(* CODESYS project Plc_CHALET_Nc.library
   Placeholder: CHALET_Nc
   Title: CHALET_Nc
   Version: 3.4.2
   Company: Beckhoff CH

Project tree, tasks and I/O mapping:
  libraries: CHALET_BaseComponents, * (Beckhoff CH); Tc2_MC2, * (Beckhoff Automation GmbH); Tc2_MC2_Drive, * (Beckhoff Automation GmbH); Tc2_Standard, * (Beckhoff Automation GmbH); Tc2_System, * (Beckhoff Automation GmbH); Tc3_EventLogger, * (Beckhoff Automation GmbH); Tc3_Module, * (Beckhoff Automation GmbH)
  COMPONENTs/
    Main FB/
      function block FB_NcAxis [ST]: Mapped, NcAxisName, NcAxisType, NcDriveType, NetId, OID, Port, GearIn, GearOut, Homing, HomingSensor, LockNegativeDirection, LockPositiveDirection, MoveAbsolute, MoveRelative, MoveVelocity, MultiGearIn, PowerOff, PowerOn, Reset, SetActPosition, Stop, ActAcceleration, ActPosition, ActPosModulo, ActVelocity, DefaultAcceleration, DefaultDeceleration, DefaultJerk, DefaultVelocity, Override, SetAcceleration, SetPosition, SetPosModulo, SetVelocity, BufferEmpty, Coupled, Enabled, Feedback, LagDistance, MotionState, Moving, FB_init, Initialize, Initialized, Prepare, Update
      interface I_AxisStatus: Override, SetAcceleration, SetPosition, SetPosModulo, SetVelocity, Enabled, LagDistance, LockNegativeDirection, LockPositiveDirection, Mapped, MotionState, Feedback, Initialized
      interface I_NcAxis_HMI: Coupled, LUID, Moving, NcAxisName
      interface I_NcAxis_PLC: GearIn, GearOut, Homing, LockNegativeDirection, LockPositiveDirection, MoveAbsolute, MoveRelative, MoveVelocity, MultiGearIn, PowerOff, PowerOn, Reset, SetActPosition, Stop, ActAcceleration, ActPosition, ActPosModulo, ActVelocity, DefaultAcceleration, DefaultDeceleration, DefaultJerk, DefaultVelocity, Override, BufferEmpty, NcAxisType, NcDriveType, Initialize, Update
    Optional/
      Adapter AXIS_REF/
        function block FB_Adapter_AXIS_REF [ST]: getAxisRef
        interface I_Adapter_AXIS_REF: getAxisRef
      Adapter HMI/
        function block FB_NcAxis_Hmi [ST]: FB_init, Update
      Casting/
        function ToNcAxisHMI [ST]
        function ToNcAxisPLC [ST]
      Feedback/
        function block FB_NcFeedback [ST]: UpdateEventlogger
      Reset/
        function block FB_Reset_NC_Sercos_CANopen [ST]
      SetActPosition/
        old/
          function block FB_SetPosition_NC_Sercos_CANopen [ST]: SetPosCoE, SetPosNC, SetPosSoE
        function block FB_SetPosition_Beckhoff [ST]
    data type E_NcAxisCommands
    NcAxisFB
  00000000-0000-0000-0000-000000000000|LICENSE.md
  LICENSE.md
  global variables NcParameterlist
*)

// COMPONENTs/E_NcAxisCommands
{attribute 'strict'}
{attribute 'to_string'}
TYPE E_NcAxisCommands :
(
	None:=0,
	Initialize,
	Reset,
	PowerOn,
	PowerOff,
	SetPosition,
	Stop,
	MoveVelocity,
	MoveRelative,
	MoveAbsolute,
	GearIn,
	GearOut,
	MultiGearIn,
	Homing,
	
	//Commands that are not handled within the basic module and must be implemented externally
	TorqueControl:=100,
	Halt,
	Jog,
	GearInDyn,
	MoveModulo,
	HaltPhasing,
	PhasingAbsolute,
	PhasingRelative,
	MoveContinuousAbsolute,
	MoveContinuousRelative,
	MoveSuperImposed,
	AbortSuperposition,
	MoveAbsoluteCA,
	MoveRelativeCA,
	HaltCA,
	GearInPosCA,
	StartExternalSetpoint,
	StopExternalSetpoint,
	
	//xPlanar
	Enable,
	Disable,
	AddToGroupe,
	RemoveFromGroupe,
	Configure,
	MoveA,
	MoveB,
	MoveC,
	MoveXY,
	MoveZ,
	JoinTrack,
	MoveOnTrack,
	Clear,
	LowerToUnknownLevel,
	LiftFromUnknownLevel,
	
	
	//Reserve
	ExternalCommand00:=200,	
	ExternalCommand01,
	ExternalCommand02,
	ExternalCommand03,
	ExternalCommand04,
	ExternalCommand05,
	ExternalCommand06,
	ExternalCommand07,
	ExternalCommand08,
	ExternalCommand09,
	ExternalCommand10,	
	ExternalCommand11,
	ExternalCommand12,
	ExternalCommand13,
	ExternalCommand14,
	ExternalCommand15,
	ExternalCommand16,
	ExternalCommand17,
	ExternalCommand18,
	ExternalCommand19

//default is none	
) := None;
END_TYPE

// NcParameterlist
{attribute 'qualified_only'}
VAR_GLOBAL CONSTANT
	ERROR_IF_NC_AXIS_IS_NOT_MAPPED : BOOL := TRUE;
END_VAR

// COMPONENTs/Main FB/FB_NcAxis
// The warning " Interface of overridden methode xxx of base I_xxx doesn't match declaration" can be disabled here. 
{warning disable C0094 }
{attribute 'no_explicit_call' := '[FB_NcAxis] Do not call the body - Stick to OOP'}
FUNCTION_BLOCK FB_NcAxis EXTENDS FB_Adapter_AXIS_REF IMPLEMENTS I_NcAxis_PLC, I_NcAxis_HMI, I_AdsAddr
VAR
	{attribute 'hide'}
	bInitDone : BOOL;
	
	//Default Values is used if commandet jerk, acc, dec or velo is 0.
	{attribute 'hide'}
	fDefaultVelocity 		: LREAL; // Read during init from NC-Axis-Parameter(init)
	{attribute 'hide'}
	fDefaultAcceleration 	: LREAL; // Read during init from NC-Axis-Parameter(init)
	{attribute 'hide'}
	fDefaultDeceleration	: LREAL; // Read during init from NC-Axis-Parameter(init)
	{attribute 'hide'}
	fDefaultJerk 			: LREAL; // Read during init from NC-Axis-Parameter(init)	
	
	//Full axis parameter set
	{attribute 'hide'}
	stAxisParameterSet 		: TC2_MC2.ST_AxisParameterSet;
	
	//Velocity override in % for all movement commands. (0 ≤ Override ≤ 100.0)
	{attribute 'hide'}
	fOverride : LREAL := 100.0;
	//Feed enable in x direction. Only takes effect if Enable = TRUE.
	{attribute 'hide'}
	bLockNegativeDirection : BOOL := FALSE;
	{attribute 'hide'}
	bLockPositiveDirection : BOOL := FALSE;
	
	//GearIn
	{attribute 'hide'}
	ipGearMasterAxis 		: I_Adapter_AXIS_REF;

	//Multigear
	{attribute 'hide'}
	ipMultiGearMasterAxis1		: I_Adapter_AXIS_REF;
	{attribute 'hide'}
	ipMultiGearMasterAxis2		: I_Adapter_AXIS_REF;
	{attribute 'hide'}
	ipMultiGearMasterAxis3		: I_Adapter_AXIS_REF;
	{attribute 'hide'}
	ipMultiGearMasterAxis4		: I_Adapter_AXIS_REF;

	{attribute 'hide'}
	fbDummyAxisRef		: TC2_MC2.AXIS_REF; // AxisRef whitout linked Nc
	
	{attribute 'hide'}               	
	fbFeedback 			: FB_NcFeedback(ipSourceInfo := fbSourceInfo);	
	
 	{attribute 'hide'}                   	
	eActiveCommand 		: E_NcAxisCommands := E_NcAxisCommands.None;
	
	{attribute 'hide'}           	
	fbPower 			: MC_Power;
	{attribute 'hide'}
	fbStop 				: MC_Stop;
	{attribute 'hide'}
	fbHoming 			: MC_Home;
	{attribute 'hide'}
	fbReset 			: FB_Reset_NC_Sercos_CANopen; 		//MC_Reset extension. can detect sercos and can and reset all faults.
	{attribute 'hide'}
	fbSetPosition 		: FB_SetPosition_Beckhoff;	//MC_SetPosition extension. Detect sercos and can and read and use the configured store position of the position feedback.(encoder/drive/NC). Set store position in DM2.
	{attribute 'hide'}
	fbMoveRelative 		: ARRAY [0..1] OF MC_MoveRelative;//A second function block is always required to use the BufferMode. It is not possible to trigger a move function block with new parameters while it is active.
	{attribute 'hide'}
	nActiveMoveRel		: UINT; 
	{attribute 'hide'}
	fbMoveAbsolute		: ARRAY [0..1] OF MC_MoveAbsolute;//A second function block is always required to use the BufferMode. It is not possible to trigger a move function block with new parameters while it is active.
	{attribute 'hide'}
	nActiveMoveAbs		: UINT; 
	{attribute 'hide'}
	fbMoveVelocity		: ARRAY [0..1] OF MC_MoveVelocity;//A second function block is always required to use the BufferMode. It is not possible to trigger a move function block with new parameters while it is active.
	{attribute 'hide'}
	nActiveMoveVel		: UINT; 
	{attribute 'hide'}
	fbGearInMultiMaster	: MC_GearInMultiMaster;
	{attribute 'hide'}
	fbGearIn 			: MC_GearIn;
	{attribute 'hide'}
	fbGearOut 			: MC_GearOut;

	{attribute 'hide'}
	bNewBufferCommadThisCycle : BOOL; //This flag is processed in the PLC cycle when a buffered motion command is requested via method


END_VAR
{warning restore C0094}

{attribute 'monitoring':='call'}
PROPERTY Mapped : BOOL //Project is mapped to NC (NcToPlc and PlcToNc)
GET
VAR
	bNcToPlcNotMapped 	: BOOL;
	bPlcToNcNotMapped 	: BOOL;
END_VAR
bPlcToNcNotMapped := F_GetMappingStatus(ADR(THIS^.Axis.PlcToNc), SIZEOF(THIS^.Axis.PlcToNc)) <> EPlcMappingStatus.MS_Mapped;
bNcToPlcNotMapped := F_GetMappingStatus(ADR(THIS^.Axis.NcToPlc), SIZEOF(THIS^.Axis.NcToPlc)) <> EPlcMappingStatus.MS_Mapped;

Mapped := NOT bNcToPlcNotMapped AND NOT bPlcToNcNotMapped;
END_GET
END_PROPERTY

{attribute 'OPC.UA.DA.Property' := '1'}
{attribute 'monitoring':='call'}
PROPERTY NcAxisName : String(31)
GET
NcAxisName := THIS^.stAxisParameterSet.sAxisName;
END_GET
END_PROPERTY

{attribute 'OPC.UA.DA.Property' := '1'}
{attribute 'monitoring':='call'}
PROPERTY NcAxisType : Tc2_MC2.E_NcAxisType
GET
NcAxisType := THIS^.stAxisParameterSet.nAxisType;
END_GET
END_PROPERTY

{attribute 'OPC.UA.DA.Property' := '1'}
{attribute 'monitoring':='call'}
PROPERTY NcDriveType : Tc2_MC2.E_NcDriveType
GET
NcDriveType:= THIS^.Axis.DriveAddress.NcDriveType;
END_GET
END_PROPERTY

{attribute 'monitoring':='call'}
PROPERTY NetId : T_AmsNetID
GET
NetId := THIS^.Axis.DriveAddress.NetID;
END_GET
END_PROPERTY

{attribute 'monitoring':='call'}
PROPERTY OID : OTCID
GET
OID := THIS^.Axis.DriveAddress.TcAxisObjectId;
END_GET
END_PROPERTY

{attribute 'monitoring':='call'}
PROPERTY Port : WORD
GET
Port := THIS^.Axis.DriveAddress.SlaveAddress;
END_GET
END_PROPERTY

{attribute 'TcRpcEnable':='1'}
(*! 
<summary>
	Establish an axis coupling to a single master axis.
	<preliminary>
		Both axis must be in standstill to apply the coupling.
		In-motion coupling of the FB is not supported by this method.
	</preliminary>
</summary>
<description>
	The coupling is performed based on a <b>velocity</b> ratio.
	As reference the master axis <b>command</b> value is used.
	There is <b>no automatic phase compensation</b> applied.
</description> 
*)

METHOD PUBLIC GearIn  : I_CH_Feedback (*! Interface to the execution feedback *)
VAR_INPUT
	(*! Interface to a master axis *)
	ipMasterAxisAdapter : I_Adapter_AXIS_REF;

	(*! Gear ratio Numerator*)
	fRatioNumerator: LREAL;
	
	(*! Gear ratio Denominator*)
	nRatioDenominator: UINT := 1;
	
	(*! Use the default dynamics if input=0.
	The default dynamics can be read and written via property and is initialized with the default values in the NC parameter list. *)
	fAcceleration	: LREAL := 0;
	
	(*! Use the default dynamics if input=0. 
	The default dynamics can be read and written via property and is initialized with the default values in the NC parameter list. *)
	fDeceleration	: LREAL := 0;
	
	(*! Use the default dynamics if input=0. 
	The default dynamics can be read and written via property and is initialized with the default values in the NC parameter list. *)
	fJerk			: LREAL := 0;
END_VAR
IF ipMasterAxisAdapter = 0 THEN
	THIS^.fbFeedback.LastCommandAccepted	:= FALSE;
	//Error not valid Input
	
ELSIF NOT __ISVALIDREF(ipMasterAxisAdapter.getAxisRef) THEN
	THIS^.fbFeedback.LastCommandAccepted	:= FALSE;
	//Invalide ref to axis
	
ELSIF fRatioNumerator = 0 OR nRatioDenominator = 0 THEN
	THIS^.fbFeedback.LastCommandAccepted	:= FALSE;
	//Error not valid Input		
	
ELSIF THIS^.fbFeedback.Error THEN
	THIS^.fbFeedback.LastCommandAccepted	:= FALSE;
	//Error active/not ready

ELSIF ipMasterAxisAdapter.getAxisRef.Status.Moving THEN		
	THIS^.fbFeedback.LastCommandAccepted	:= FALSE;
	//Only support geraring in standstill

ELSIF THIS^.Axis.Status.Moving THEN		
	THIS^.fbFeedback.LastCommandAccepted	:= FALSE;	
	//Only support geraring in standstill

ELSE
	THIS^.eActiveCommand 				:= E_NcAxisCommands.GearIn;
	THIS^.fbFeedback.ActiveCommand 		:= TO_STRING(THIS^.eActiveCommand);
	THIS^.fbFeedback.LastCommandAccepted:= TRUE;
	THIS^.fbFeedback.Busy 				:= TRUE;
	
	THIS^.ipGearMasterAxis 				:= ipMasterAxisAdapter;
	
	THIS^.fbGearIn.Execute				:= TRUE;
	THIS^.fbGearIn.RatioNumerator 		:= fRatioNumerator;	
	THIS^.fbGearIn.RatioDenominator     := nRatioDenominator;		
	
	//Acceleration
	//If input = 0  then use default dynamics
	IF fAcceleration = 0.0 THEN
		THIS^.fbGearIn.Acceleration := THIS^.fDefaultAcceleration;
	ELSE
		THIS^.fbGearIn.Acceleration := fAcceleration;
	END_IF
	
	//Deceleration
	//If input = 0  then use default dynamics
	IF fDeceleration = 0.0 THEN
		THIS^.fbGearIn.Deceleration := THIS^.fDefaultDeceleration;
	ELSE
		THIS^.fbGearIn.Deceleration := fDeceleration;
	END_IF
	
	//Jerk
	//If input = 0  then use default dynamics
	IF fJerk = 0.0 THEN
		THIS^.fbGearIn.Jerk := THIS^.fDefaultJerk;
	ELSE
		THIS^.fbGearIn.Jerk := fJerk;
	END_IF
END_IF


GearIn := THIS^.fbFeedback;
END_METHOD

{attribute 'TcRpcEnable':='1'} 
(*WARNING
No standstill of the axis due to decoupling
When a slave axis is uncoupled during the movement, it is not stopped automatically but reaches a constant velocity at which it continues to travel infinitely.
You can stop the axis with the function blocks MC_Halt or MC_Stop.*)
METHOD GearOut  : I_CH_Feedback


THIS^.eActiveCommand 				:= E_NcAxisCommands.GearOut;
THIS^.fbFeedback.ActiveCommand 		:= TO_STRING(THIS^.eActiveCommand);
THIS^.fbFeedback.LastCommandAccepted:= TRUE;
THIS^.fbFeedback.Busy 				:= TRUE;

THIS^.fbGearOut.Execute				:= TRUE;

THIS^.ipGearMasterAxis 				:= 0;
THIS^.ipMultiGearMasterAxis1 		:= 0;
THIS^.ipMultiGearMasterAxis2 		:= 0;
THIS^.ipMultiGearMasterAxis3 		:= 0;
THIS^.ipMultiGearMasterAxis4 		:= 0;



GearOut := THIS^.fbFeedback;
END_METHOD

{attribute 'TcRpcEnable':='1'} 
(*The parameterization of the home command takes place in the NC! To do this, set the parameters in:
- NC-Axis(Parameters) Homing speed
- NC-Axis>Encoder(Parameters) Homing mode
	Reference Mode: "Homing Sensor Only"
	Homing Sensor Source "Digital Input x" 
		Link Input to NC-Axis>Drive>Inputs>nState8.x
		
The "HomeingSensor" property can also be used to control a home sensor via PLC.		
*)
(*Homing refers to an axis initialization run during which the correct actual position is determined by means of a reference signal. This can be NC-guided, as default described here:
  - The axis is at a random position.
  - The axis moves in the parameterized direction and searches for the reference switch (referencing cam/calibration cam).
  - The axis reverses as soon as the referencing cam is detected.
  - The axis moves away from the referencing cam and detects the falling edge of the cam signal.
  - The reference position is set and the axis stops. The standstill position of the axis deviates slightly from the reference position.*)
METHOD Homing  : I_CH_Feedback
VAR_INPUT
	(*Absolute reference position to which the axis is set after homing*)
	fPosition		: LREAL;
END_VAR
IF THIS^.fbFeedback.Error THEN
	THIS^.fbFeedback.LastCommandAccepted	:= FALSE;
	//Error active/not ready

ELSIF NOT THIS^.BufferEmpty THEN		
	THIS^.fbFeedback.LastCommandAccepted	:= FALSE;
	//Buffer not ready to store next motion command	
	
ELSIF NOT(THIS^.Axis.Status.StandStill OR THIS^.Axis.Status.DiscreteMotion OR THIS^.Axis.Status.ContinuousMotion OR THIS^.Axis.Status.SynchronizedMotion) THEN		
	THIS^.fbFeedback.LastCommandAccepted	:= FALSE;
	//Axis in wrong State

	
ELSE
	THIS^.eActiveCommand 				:= E_NcAxisCommands.Homing;
	THIS^.fbFeedback.ActiveCommand 		:= TO_STRING(THIS^.eActiveCommand);
	THIS^.fbFeedback.LastCommandAccepted:= TRUE;                                  
	THIS^.fbFeedback.Busy 				:= TRUE;
	                                    
	THIS^.fbHoming.Execute				:= TRUE;
	 (* default homing as defined in the SystemManager encoder parameters *)
	THIS^.fbHoming.HomingMode			:= MC_HomingMode.MC_DefaultHoming;
	
	THIS^.fbHoming.Position				:= fPosition;
	
END_IF


Homing := THIS^.fbFeedback;
END_METHOD

//A home input switch can be linked here. Whether this works depends heavily on how the settings in the NC2-axis and NC2-axis-encoder are configured.
PROPERTY HomingSensor : BOOL
SET
THIS^.fbHoming.bCalibrationCam := HomingSensor;
END_SET
END_PROPERTY

{attribute 'monitoring':='call'}
//Disable the feed in one direction.
PROPERTY LockNegativeDirection : BOOL
GET
LockNegativeDirection := bLockNegativeDirection;
END_GET
SET
VAR_INST
	{attribute 'hide'}
	fbInfoFeedDisabled : FB_TcAlarm;
END_VAR
THIS^.bLockNegativeDirection := LockNegativeDirection;


//Creat an info in TC3_Eventlogger
IF NOT fbInfoFeedDisabled.bRaised AND THIS^.bLockNegativeDirection THEN
	fbInfoFeedDisabled.CreateEx(stEventEntry := TC_EVENTS.CHALET_NC_Events.FeedNegativeDisabled, bWithConfirmation := FALSE, ipSourceInfo := THIS^.fbSourceInfo);
	fbInfoFeedDisabled.Raise(0);
	
ELSIF NOT THIS^.bLockNegativeDirection THEN
	fbInfoFeedDisabled.Clear(0, 0);
END_IF
END_SET
END_PROPERTY

{attribute 'monitoring':='call'}
//Disable the feed in one direction.
PROPERTY LockPositiveDirection : BOOL
GET
LockPositiveDirection := bLockPositiveDirection;
END_GET
SET
VAR_INST
	{attribute 'hide'}
	fbInfoFeedDisabled : FB_TcAlarm;
END_VAR
THIS^.bLockPositiveDirection := LockPositiveDirection;


//Creat an info in TC3_Eventlogger
IF NOT fbInfoFeedDisabled.bRaised AND THIS^.bLockPositiveDirection THEN
	fbInfoFeedDisabled.CreateEx(stEventEntry := TC_EVENTS.CHALET_NC_Events.FeedPositiveDisabled, bWithConfirmation := FALSE, ipSourceInfo := THIS^.fbSourceInfo);
	fbInfoFeedDisabled.Raise(0);
	
ELSIF NOT THIS^.bLockPositiveDirection THEN
	fbInfoFeedDisabled.Clear(0, 0);
END_IF
END_SET
END_PROPERTY

{attribute 'TcRpcEnable':='1'} 
METHOD MoveAbsolute  : I_CH_Feedback
VAR_INPUT
	fPosition		: LREAL;
	
	(* Use the default dynamics if input=0. 
	The default dynamics can be read and written via property and is initialized with the default values in the NC parameter list. *)
	fVelocity		: LREAL := 0;
	
	(* Use the default dynamics if input=0. 
	The default dynamics can be read and written via property and is initialized with the default values in the NC parameter list. *)
	fAcceleration	: LREAL := 0;
	
	(* Use the default dynamics if input=0. 
	The default dynamics can be read and written via property and is initialized with the default values in the NC parameter list. *)
	fDeceleration	: LREAL := 0;
	
	(* Use the default dynamics if input=0. 
	The default dynamics can be read and written via property and is initialized with the default values in the NC parameter list. *)
	fJerk			: LREAL := 0;
	
	(* Input=0 = MC_Aborting   
	BufferModes:
		-MC_Aborting: Default mode without buffering. The command is executed immediately and interrupts any other command that may be running.
		-MC_Buffered: The command is executed once no other command is running on the axis. The previous movement continues until it has stopped. The following command is started from standstill.
		-MC_BlendingLow: The command is executed once no other command is running on the axis. In contrast to Buffered the axis does not stop at the previous target, but passes through this position with the lower velocity of two commands.
		-MC_BlendingHigh The command is executed once no other command is running on the axis. In contrast to Buffered the axis does not stop at the previous target, but passes through this position with the higher velocity of two commands.
		-MC_BlendingNext: The command is executed once no other command is running on the axis. In contrast to Buffered the axis does not stop at the previous target, but passes through this position with the velocity of the last command.
		-MC_BlendingPrevious: The command is executed once no other command is running on the axis. In contrast to Buffered the axis does not stop at the previous target, but passes through this position with the velocity of the first command. *)
	eBufferMode   : Tc2_MC2.MC_BufferMode := Tc2_MC2.MC_BufferMode.MC_Aborting;
END_VAR
VAR
	nInactiveInstance : UINT;
END_VAR
IF THIS^.fbFeedback.Error THEN
	THIS^.fbFeedback.LastCommandAccepted	:= FALSE;
	//Error active/not ready

ELSIF NOT THIS^.BufferEmpty THEN		
	THIS^.fbFeedback.LastCommandAccepted	:= FALSE;
	//Buffer not ready to store next motion command	
	
ELSIF NOT(THIS^.Axis.Status.StandStill OR THIS^.Axis.Status.DiscreteMotion OR THIS^.Axis.Status.ContinuousMotion OR THIS^.Axis.Status.SynchronizedMotion) THEN		
	THIS^.fbFeedback.LastCommandAccepted	:= FALSE;
	//Axis in wrong State
	
ELSIF (eBufferMode <> MC_BufferMode.MC_Aborting) AND bNewBufferCommadThisCycle THEN		
	THIS^.fbFeedback.LastCommandAccepted	:= FALSE;
	//Buffer not ready to store next motion command		
	//Max send one buffered motion command each cycle	
	
ELSE
	//A second function block is always required to use the BufferMode. It is not possible to trigger a move function block with new parameters while it is active.
	IF THIS^.fbMoveAbsolute[nActiveMoveAbs].Busy THEN
		nInactiveInstance := (THIS^.nActiveMoveAbs + 1)MOD 2;
	ELSE
		nInactiveInstance := THIS^.nActiveMoveAbs;
	END_IF
	
	THIS^.eActiveCommand 				:= E_NcAxisCommands.MoveAbsolute;
	THIS^.fbFeedback.ActiveCommand 		:= TO_STRING(THIS^.eActiveCommand);
	THIS^.fbFeedback.LastCommandAccepted:= TRUE;		
	THIS^.fbFeedback.Busy 				:= TRUE;
	
	THIS^.fbMoveAbsolute[nInactiveInstance].Execute		:= TRUE;
	THIS^.fbMoveAbsolute[nInactiveInstance].Position	:= fPosition;
	THIS^.fbMoveAbsolute[nInactiveInstance].BufferMode 	:= eBufferMode;
	
	//If the currend command is a buffered movement, then set a flag.
	IF eBufferMode <> MC_BufferMode.MC_Aborting THEN
		THIS^.bNewBufferCommadThisCycle := TRUE;
	END_IF
	
	//Velocity
	//If input = 0  then use default dynamics
	IF fVelocity = 0.0 THEN
		THIS^.fbMoveAbsolute[nInactiveInstance].Velocity := THIS^.fDefaultVelocity;
	ELSE
		THIS^.fbMoveAbsolute[nInactiveInstance].Velocity := fVelocity;
	END_IF
	
	//Acceleration
	//If input = 0  then use default dynamics
	IF fAcceleration = 0.0 THEN
		THIS^.fbMoveAbsolute[nInactiveInstance].Acceleration := THIS^.fDefaultAcceleration;
	ELSE
		THIS^.fbMoveAbsolute[nInactiveInstance].Acceleration := fAcceleration;
	END_IF
	
	//Deceleration
	//If input = 0  then use default dynamics
	IF fDeceleration = 0.0 THEN
		THIS^.fbMoveAbsolute[nInactiveInstance].Deceleration := THIS^.fDefaultDeceleration;
	ELSE
		THIS^.fbMoveAbsolute[nInactiveInstance].Deceleration := fDeceleration;
	END_IF
	
	//Jerk
	//If input = 0  then use default dynamics
	IF fJerk = 0.0 THEN
		THIS^.fbMoveAbsolute[nInactiveInstance].Jerk := THIS^.fDefaultJerk;
	ELSE
		THIS^.fbMoveAbsolute[nInactiveInstance].Jerk := fJerk;
	END_IF

END_IF


MoveAbsolute := THIS^.fbFeedback;
END_METHOD

{attribute 'TcRpcEnable':='1'} 
METHOD MoveRelative  : I_CH_Feedback
VAR_INPUT
	fDistance		: LREAL;
	
	(* Use the default dynamics if input=0. 
	The default dynamics can be read and written via property and is initialized with the default values in the NC parameter list. *)
	fVelocity		: LREAL := 0;
	
	(* Use the default dynamics if input=0. 
	The default dynamics can be read and written via property and is initialized with the default values in the NC parameter list. *)
	fAcceleration	: LREAL := 0;
	
	(* Use the default dynamics if input=0. 
	The default dynamics can be read and written via property and is initialized with the default values in the NC parameter list. *)
	fDeceleration	: LREAL := 0;
	
	(* Use the default dynamics if input=0. 
	The default dynamics can be read and written via property and is initialized with the default values in the NC parameter list. *)
	fJerk			: LREAL := 0;
	
	(* Input=0 = MC_Aborting   
	BufferModes:
		-MC_Aborting: Default mode without buffering. The command is executed immediately and interrupts any other command that may be running.
		-MC_Buffered: The command is executed once no other command is running on the axis. The previous movement continues until it has stopped. The following command is started from standstill.
		-MC_BlendingLow: The command is executed once no other command is running on the axis. In contrast to Buffered the axis does not stop at the previous target, but passes through this position with the lower velocity of two commands.
		-MC_BlendingHigh The command is executed once no other command is running on the axis. In contrast to Buffered the axis does not stop at the previous target, but passes through this position with the higher velocity of two commands.
		-MC_BlendingNext: The command is executed once no other command is running on the axis. In contrast to Buffered the axis does not stop at the previous target, but passes through this position with the velocity of the last command.
		-MC_BlendingPrevious: The command is executed once no other command is running on the axis. In contrast to Buffered the axis does not stop at the previous target, but passes through this position with the velocity of the first command. *)
	eBufferMode   : Tc2_MC2.MC_BufferMode := Tc2_MC2.MC_BufferMode.MC_Aborting;
END_VAR
VAR
	nInactiveInstance : UINT;
END_VAR
IF THIS^.fbFeedback.Error THEN
	THIS^.fbFeedback.LastCommandAccepted	:= FALSE;
	//Error active/not ready

ELSIF NOT THIS^.BufferEmpty THEN		
	THIS^.fbFeedback.LastCommandAccepted	:= FALSE;
	//Buffer not ready to store next motion command	
	
ELSIF NOT(THIS^.Axis.Status.StandStill OR THIS^.Axis.Status.DiscreteMotion OR THIS^.Axis.Status.ContinuousMotion OR THIS^.Axis.Status.SynchronizedMotion) THEN		
	THIS^.fbFeedback.LastCommandAccepted	:= FALSE;
	//Axis in wrong State

ELSIF (eBufferMode <> MC_BufferMode.MC_Aborting) AND bNewBufferCommadThisCycle THEN		
	THIS^.fbFeedback.LastCommandAccepted	:= FALSE;
	//Buffer not ready to store next motion command		
	//Max send one buffered motion command each cycle	
		
	
//ZZZ Todo Bug in 4024, only allow buffered movement if an 'normal' movement is active.	
ELSIF (eBufferMode <> MC_BufferMode.MC_Aborting) AND NOT THIS^.Axis.Status.HasJob THEN		
	THIS^.fbFeedback.LastCommandAccepted	:= FALSE;
	//Buffered movement not possible if axis is not moving
	
ELSE
	//A second function block is always required to use the BufferMode. It is not possible to trigger a move function block with new parameters while it is active.
	IF THIS^.fbMoveRelative[nActiveMoveRel].Busy THEN
		nInactiveInstance := (THIS^.nActiveMoveRel + 1)MOD 2;
	ELSE
		nInactiveInstance := THIS^.nActiveMoveRel;
	END_IF

	THIS^.eActiveCommand 				:= E_NcAxisCommands.MoveRelative;
	THIS^.fbFeedback.ActiveCommand 		:= TO_STRING(THIS^.eActiveCommand);
	THIS^.fbFeedback.LastCommandAccepted:= TRUE;                                  
	THIS^.fbFeedback.Busy 				:= TRUE;
	                                    
	THIS^.fbMoveRelative[nInactiveInstance].Execute		:= TRUE;
	THIS^.fbMoveRelative[nInactiveInstance].Distance	:= fDistance;
	THIS^.fbMoveRelative[nInactiveInstance].BufferMode 	:= eBufferMode;
	
	//If the currend command is a buffered movement, then set a flag.
	IF eBufferMode <> MC_BufferMode.MC_Aborting THEN
		THIS^.bNewBufferCommadThisCycle := TRUE;
	END_IF
	
	//Velocity
	//If input = 0  then use default dynamics
	IF fVelocity = 0.0 THEN
		THIS^.fbMoveRelative[nInactiveInstance].Velocity := THIS^.fDefaultVelocity;
	ELSE
		THIS^.fbMoveRelative[nInactiveInstance].Velocity := fVelocity;
	END_IF
	
	//Acceleration
	//If input = 0  then use default dynamics
	IF fAcceleration = 0.0 THEN
		THIS^.fbMoveRelative[nInactiveInstance].Acceleration := THIS^.fDefaultAcceleration;
	ELSE
		THIS^.fbMoveRelative[nInactiveInstance].Acceleration := fAcceleration;
	END_IF
	
	//Deceleration
	//If input = 0  then use default dynamics
	IF fDeceleration = 0.0 THEN
		THIS^.fbMoveRelative[nInactiveInstance].Deceleration := THIS^.fDefaultDeceleration;
	ELSE
		THIS^.fbMoveRelative[nInactiveInstance].Deceleration := fDeceleration;
	END_IF
	
	//Jerk
	//If input = 0  then use default dynamics
	IF fJerk = 0.0 THEN
		THIS^.fbMoveRelative[nInactiveInstance].Jerk := THIS^.fDefaultJerk;
	ELSE
		THIS^.fbMoveRelative[nInactiveInstance].Jerk := fJerk;
	END_IF
END_IF


MoveRelative := THIS^.fbFeedback;
END_METHOD

{attribute 'TcRpcEnable':='1'} 
METHOD MoveVelocity  : I_CH_Feedback
VAR_INPUT
	(* Use the default dynamics if input=0. 
	The default dynamics can be read and written via property and is initialized with the default values in the NC parameter list. *)
	fVelocity		: LREAL:= 0;
	
	(* Use the default dynamics if input=0. 
	The default dynamics can be read and written via property and is initialized with the default values in the NC parameter list. *)
	fAcceleration	: LREAL := 0;
	
	(* Use the default dynamics if input=0. 
	The default dynamics can be read and written via property and is initialized with the default values in the NC parameter list. *)
	fDeceleration	: LREAL := 0;
	
	(* Use the default dynamics if input=0. 
	The default dynamics can be read and written via property and is initialized with the default values in the NC parameter list. *)
	fJerk			: LREAL := 0;
	
	(* If input=1, then direction is positive. 
	Positive OR negative direction of travel (TYPE: Tc2_MC2.MC_Direction) *)
	eDirection: Tc2_MC2.MC_Direction := Tc2_MC2.MC_Direction.MC_Positive_Direction;
	
	(* Input=0 = MC_Aborting   
	BufferModes:
		-MC_Aborting: Default mode without buffering. The command is executed immediately and interrupts any other command that may be running.
		-MC_Buffered: The command is executed once no other command is running on the axis. The previous movement continues until it has stopped. The following command is started from standstill.
		-MC_BlendingLow: The command is executed once no other command is running on the axis. In contrast to Buffered the axis does not stop at the previous target, but passes through this position with the lower velocity of two commands.
		-MC_BlendingHigh The command is executed once no other command is running on the axis. In contrast to Buffered the axis does not stop at the previous target, but passes through this position with the higher velocity of two commands.
		-MC_BlendingNext: The command is executed once no other command is running on the axis. In contrast to Buffered the axis does not stop at the previous target, but passes through this position with the velocity of the last command.
		-MC_BlendingPrevious: The command is executed once no other command is running on the axis. In contrast to Buffered the axis does not stop at the previous target, but passes through this position with the velocity of the first command. *)
	eBufferMode   : Tc2_MC2.MC_BufferMode := Tc2_MC2.MC_BufferMode.MC_Aborting;;
END_VAR
VAR
	nInactiveInstance : UINT;
END_VAR
IF THIS^.fbFeedback.Error THEN
	THIS^.fbFeedback.LastCommandAccepted	:= FALSE;
	//Error active/not ready

ELSIF NOT THIS^.BufferEmpty THEN		
	THIS^.fbFeedback.LastCommandAccepted	:= FALSE;
	//Buffer not ready to store next motion command	
	
ELSIF NOT(THIS^.Axis.Status.StandStill OR THIS^.Axis.Status.DiscreteMotion OR THIS^.Axis.Status.ContinuousMotion OR THIS^.Axis.Status.SynchronizedMotion) THEN		
	THIS^.fbFeedback.LastCommandAccepted	:= FALSE;
	//Axis in wrong State

ELSIF (eBufferMode <> MC_BufferMode.MC_Aborting) AND bNewBufferCommadThisCycle THEN		
	THIS^.fbFeedback.LastCommandAccepted	:= FALSE;
	//Buffer not ready to store next motion command		
	//Max send one buffered motion command each cycle	
	
	
ELSE
	//A second function block is always required to use the BufferMode. It is not possible to trigger a move function block with new parameters while it is active.
	IF THIS^.fbMoveVelocity[nActiveMoveVel].Busy THEN
		nInactiveInstance := (THIS^.nActiveMoveVel + 1)MOD 2;
	ELSE
		nInactiveInstance := THIS^.nActiveMoveVel;
	END_IF
	
	//Direction 0 is not an valide enumeration. If input=0, then default direction is positive
	IF eDirection = 0 THEN
		eDirection := Tc2_MC2.MC_Direction.MC_Positive_Direction;
	END_IF
	
	THIS^.eActiveCommand 				:= E_NcAxisCommands.MoveVelocity;	
	THIS^.fbFeedback.ActiveCommand 		:= TO_STRING(THIS^.eActiveCommand);
	THIS^.fbFeedback.LastCommandAccepted:= TRUE;	
	THIS^.fbFeedback.Busy 				:= TRUE;
	
	THIS^.fbMoveVelocity[nInactiveInstance].Execute		:= TRUE;	
	THIS^.fbMoveVelocity[nInactiveInstance].Direction		:= eDirection; 	
	THIS^.fbMoveVelocity[nInactiveInstance].BufferMode		:= eBufferMode; 	
	
	//If the currend command is a buffered movement, then set a flag.
	IF eBufferMode <> MC_BufferMode.MC_Aborting THEN
		THIS^.bNewBufferCommadThisCycle := TRUE;
	END_IF
	
	//Velocity
	//If input = 0  then use default dynamics
	IF fVelocity = 0.0 THEN
		THIS^.fbMoveVelocity[nInactiveInstance].Velocity := THIS^.fDefaultVelocity;
	ELSE
		THIS^.fbMoveVelocity[nInactiveInstance].Velocity := fVelocity;
	END_IF
	
	//Acceleration
	//If input = 0  then use default dynamics
	IF fAcceleration = 0.0 THEN
		THIS^.fbMoveVelocity[nInactiveInstance].Acceleration := THIS^.fDefaultAcceleration;
	ELSE
		THIS^.fbMoveVelocity[nInactiveInstance].Acceleration := fAcceleration;
	END_IF
	
	//Deceleration
	//If input = 0  then use default dynamics
	IF fDeceleration = 0.0 THEN
		THIS^.fbMoveVelocity[nInactiveInstance].Deceleration := THIS^.fDefaultDeceleration;
	ELSE
		THIS^.fbMoveVelocity[nInactiveInstance].Deceleration := fDeceleration;
	END_IF
	
	//Jerk
	//If input = 0  then use default dynamics
	IF fJerk = 0.0 THEN
		THIS^.fbMoveVelocity[nInactiveInstance].Jerk := THIS^.fDefaultJerk;
	ELSE
		THIS^.fbMoveVelocity[nInactiveInstance].Jerk := fJerk;
	END_IF
END_IF


MoveVelocity := THIS^.fbFeedback;
END_METHOD

{attribute 'TcRpcEnable':='1'} 
METHOD MultiGearIn : I_CH_Feedback
VAR_INPUT
	(* Interface to an master axis *)
	ipMasterAxisAdapter : I_Adapter_AXIS_REF;
	
	(* Gear ratio Numerator*)
	fRatioNumerator: LREAL;
	(* Gear ratio Denominator*)
	nRatioDenominator: UINT := 1;
	
	(* Use the default dynamics if input=0. 
	The default dynamics can be read and written via property and is initialized with the default values in the NC parameter list. *)
	fAcceleration	: LREAL := 0;
	
	(* Use the default dynamics if input=0. 
	The default dynamics can be read and written via property and is initialized with the default values in the NC parameter list. *)
	fDeceleration	: LREAL := 0;
	
	(* Use the default dynamics if input=0. 
	The default dynamics can be read and written via property and is initialized with the default values in the NC parameter list. *)
	fJerk			: LREAL := 0;
END_VAR
IF ipMasterAxisAdapter = 0 THEN
	THIS^.fbFeedback.LastCommandAccepted	:= FALSE;
	//Error not valid Input
	
ELSIF NOT __ISVALIDREF(ipMasterAxisAdapter.getAxisRef) THEN
	THIS^.fbFeedback.LastCommandAccepted	:= FALSE;
	//Invalide ref to axis
	
ELSIF fRatioNumerator = 0 OR nRatioDenominator = 0 THEN
	THIS^.fbFeedback.LastCommandAccepted	:= FALSE;
	//Error not valid Input	

ELSIF THIS^.fbFeedback.Error THEN
	THIS^.fbFeedback.LastCommandAccepted	:= FALSE;
	//Error active/not ready

ELSIF ipMasterAxisAdapter.getAxisRef.Status.Moving THEN		
	THIS^.fbFeedback.LastCommandAccepted	:= FALSE;
	//Only support geraring in standstill

ELSIF THIS^.Axis.Status.Moving THEN		
	THIS^.fbFeedback.LastCommandAccepted	:= FALSE;	
	//Only support geraring in standstill
	
ELSE
	THIS^.eActiveCommand 					:= E_NcAxisCommands.MultiGearIn;
	THIS^.fbFeedback.ActiveCommand 		:= TO_STRING(THIS^.eActiveCommand);
	THIS^.fbFeedback.LastCommandAccepted	:= TRUE;
	THIS^.fbFeedback.Busy 					:= TRUE;
	
	IF (THIS^.ipMultiGearMasterAxis1=0) OR (THIS^.ipMultiGearMasterAxis1=ipMasterAxisAdapter) THEN
		THIS^.ipMultiGearMasterAxis1 				:= ipMasterAxisAdapter;
		THIS^.fbGearInMultiMaster.GearRatio1 		:= (fRatioNumerator/nRatioDenominator);
	ELSIF (THIS^.ipMultiGearMasterAxis2=0) OR (THIS^.ipMultiGearMasterAxis2=ipMasterAxisAdapter)  THEN
		THIS^.ipMultiGearMasterAxis2 				:= ipMasterAxisAdapter;
		THIS^.fbGearInMultiMaster.GearRatio2 		:= (fRatioNumerator/nRatioDenominator);
	ELSIF (THIS^.ipMultiGearMasterAxis3=0) OR (THIS^.ipMultiGearMasterAxis3=ipMasterAxisAdapter)  THEN
		THIS^.ipMultiGearMasterAxis3 				:= ipMasterAxisAdapter;
		THIS^.fbGearInMultiMaster.GearRatio3 		:= (fRatioNumerator/nRatioDenominator);
	ELSIF (THIS^.ipMultiGearMasterAxis4=0) OR (THIS^.ipMultiGearMasterAxis4=ipMasterAxisAdapter)  THEN
		THIS^.ipMultiGearMasterAxis4 				:= ipMasterAxisAdapter;
		THIS^.fbGearInMultiMaster.GearRatio4 		:= (fRatioNumerator/nRatioDenominator);
	ELSE
		//List is full. Only Multigeat up to 4 axis
		;
	END_IF

	
	// Open existing gear to couple a new
	THIS^.fbGearOut.Execute		:= TRUE;
	
	//Acceleration
	//If input = 0  then use default dynamics
	IF fAcceleration = 0.0 THEN
		THIS^.fbGearInMultiMaster.Acceleration := THIS^.fDefaultAcceleration;
	ELSE
		THIS^.fbGearInMultiMaster.Acceleration := fAcceleration;
	END_IF
	
	//Deceleration
	//If input = 0  then use default dynamics
	IF fDeceleration = 0.0 THEN
		THIS^.fbGearInMultiMaster.Deceleration := THIS^.fDefaultDeceleration;
	ELSE
		THIS^.fbGearInMultiMaster.Deceleration := fDeceleration;
	END_IF
	
	//Jerk
	//If input = 0  then use default dynamics
	IF fJerk = 0.0 THEN
		THIS^.fbGearInMultiMaster.Jerk := THIS^.fDefaultJerk;
	ELSE
		THIS^.fbGearInMultiMaster.Jerk := fJerk;
	END_IF
END_IF



MultiGearIn := THIS^.fbFeedback;
END_METHOD

{attribute 'TcRpcEnable':='1'} 
METHOD PowerOff  : I_CH_Feedback
//No IF. Allways allow to disable the power
THIS^.eActiveCommand 				:= E_NcAxisCommands.PowerOff;	
THIS^.fbFeedback.ActiveCommand 		:= TO_STRING(THIS^.eActiveCommand);
THIS^.fbFeedback.LastCommandAccepted:= TRUE;
THIS^.fbFeedback.Busy 				:= TRUE;	

THIS^.fbPower.Enable				:= FALSE;


PowerOff := THIS^.fbFeedback;
END_METHOD

{attribute 'TcRpcEnable':='1'} 
METHOD PowerOn : I_CH_Feedback
IF NOT (THIS^.fbFeedback.HR = S_OK) THEN
	THIS^.fbFeedback.LastCommandAccepted	:= FALSE;
	//Error active/not ready

ELSIF NOT(THIS^.Axis.Status.Disabled) THEN	
	THIS^.fbFeedback.LastCommandAccepted	:= FALSE;	
	//Axis in wrong State
	
ELSE
	THIS^.eActiveCommand 				:= E_NcAxisCommands.PowerOn; 
	THIS^.fbFeedback.ActiveCommand 		:= TO_STRING(THIS^.eActiveCommand);    
	THIS^.fbFeedback.LastCommandAccepted:= TRUE;                        	
	THIS^.fbFeedback.Busy 				:= TRUE;
	                                	
	THIS^.fbPower.Enable				:= TRUE;
	THIS^.fbPower.Enable_Positive		:= TRUE;
	THIS^.fbPower.Enable_Negative		:= TRUE;
END_IF



PowerOn := THIS^.fbFeedback;
END_METHOD

{attribute 'TcRpcEnable':='1'} 
METHOD Reset : I_CH_Feedback
THIS^.eActiveCommand 				:= E_NcAxisCommands.Reset;	
THIS^.fbFeedback.ActiveCommand 		:= TO_STRING(THIS^.eActiveCommand);
THIS^.fbFeedback.LastCommandAccepted:= TRUE;
THIS^.fbFeedback.Busy 				:= TRUE;

THIS^.fbReset.Execute				:= TRUE;


Reset := THIS^.fbFeedback;
END_METHOD

{attribute 'TcRpcEnable':='1'} 
//Set the current position of the axis to a new value. However, this is only temporary until the next restart in the NC.
METHOD SetActPosition : I_CH_Feedback
VAR_INPUT
	fPosition: LREAL;//Absolute
END_VAR
IF NOT(THIS^.Axis.Status.StandStill OR THIS^.Axis.Status.Disabled OR THIS^.Axis.Status.ErrorStop) THEN	
	THIS^.fbFeedback.LastCommandAccepted	:= FALSE;	
	//Axis in wrong State
	//zzz todo set error 33105
	
ELSIF THIS^.Axis.Status.Coupled THEN	
	THIS^.fbFeedback.LastCommandAccepted	:= FALSE;	
	//Axis is in gear
	
ELSE
	THIS^.eActiveCommand 					:= E_NcAxisCommands.SetPosition;
	THIS^.fbFeedback.ActiveCommand 			:= TO_STRING(THIS^.eActiveCommand);
	THIS^.fbFeedback.LastCommandAccepted	:= TRUE;
	THIS^.fbFeedback.Busy 					:= TRUE;
	                                    	
	THIS^.fbSetPosition.Execute				:= TRUE;
	THIS^.fbSetPosition.Position			:= fPosition;	
	THIS^.fbSetPosition.Mode				:= FALSE;	//FALSE=Absolute	
END_IF


SetActPosition := THIS^.fbFeedback;
END_METHOD

{attribute 'TcRpcEnable':='1'}
//The .Stop() is used to stop an axis with a defined deceleration ramp. Abort of all movement commands
METHOD Stop : I_CH_Feedback
VAR_INPUT
	(* Use the default dynamics if input=0. 
	The default dynamics can be read and written via property and is initialized with the default values in the NC parameter list. *)
	fDeceleration: LREAL := 0;
	
	(* Use the default dynamics if input=0. 
	The default dynamics can be read and written via property and is initialized with the default values in the NC parameter list. *)
	fJerk: LREAL := 0;
END_VAR
//No IF. Allways allow to stop the ax
THIS^.eActiveCommand 				:= E_NcAxisCommands.Stop;
THIS^.fbFeedback.ActiveCommand 		:= TO_STRING(THIS^.eActiveCommand);
THIS^.fbFeedback.LastCommandAccepted:= TRUE;
THIS^.fbFeedback.Busy 				:= TRUE;	

THIS^.fbStop.Execute				:= TRUE;

//open gear
THIS^.ipGearMasterAxis 				:= 0;
THIS^.ipMultiGearMasterAxis1 		:= 0;
THIS^.ipMultiGearMasterAxis2 		:= 0;
THIS^.ipMultiGearMasterAxis3 		:= 0;
THIS^.ipMultiGearMasterAxis4 		:= 0;
	
//Deceleration
//If input = 0  then use default dynamics
IF fDeceleration = 0.0 THEN
	THIS^.fbStop.Deceleration := THIS^.fDefaultDeceleration;
ELSE
	THIS^.fbStop.Deceleration := fDeceleration;
END_IF

//Jerk
//If input = 0  then use default dynamics
IF fJerk = 0.0 THEN
	THIS^.fbStop.Jerk := THIS^.fDefaultJerk;
ELSE
	THIS^.fbStop.Jerk := fJerk;
END_IF



Stop := THIS^.fbFeedback;
END_METHOD

{attribute 'OPC.UA.DA.Property' := '1'}
{attribute 'monitoring':='call'}
PROPERTY ActAcceleration : LREAL
GET
ActAcceleration := THIS^.Axis.NcToPlc.ActAcc;
END_GET
END_PROPERTY

{attribute 'OPC.UA.DA.Property' := '1'}
{attribute 'monitoring':='call'}
PROPERTY ActPosition : LREAL
GET
ActPosition := THIS^.Axis.NcToPlc.ActPos;
END_GET
END_PROPERTY

{attribute 'OPC.UA.DA.Property' := '1'}
{attribute 'monitoring':='call'}
PROPERTY ActPosModulo : LREAL
GET
ActPosModulo := THIS^.Axis.NcToPlc.ModuloActPos;
END_GET
END_PROPERTY

{attribute 'OPC.UA.DA.Property' := '1'}
{attribute 'monitoring':='call'}
PROPERTY ActVelocity : LREAL
GET
ActVelocity := THIS^.Axis.NcToPlc.ActVelo;
END_GET
END_PROPERTY

{attribute 'OPC.UA.DA.Property' := '1'}
{attribute 'monitoring':='call'}
PROPERTY DefaultAcceleration : LREAL
GET
DefaultAcceleration := THIS^.fDefaultAcceleration;
END_GET
SET
THIS^.fDefaultAcceleration := DefaultAcceleration;
END_SET
END_PROPERTY

{attribute 'OPC.UA.DA.Property' := '1'}
{attribute 'monitoring':='call'}
PROPERTY DefaultDeceleration : LREAL
GET
DefaultDeceleration := THIS^.fDefaultDeceleration;
END_GET
SET
THIS^.fDefaultDeceleration := DefaultDeceleration;
END_SET
END_PROPERTY

{attribute 'OPC.UA.DA.Property' := '1'}
{attribute 'monitoring':='call'}
PROPERTY DefaultJerk : LREAL
GET
DefaultJerk := THIS^.fDefaultJerk;
END_GET
SET
THIS^.fDefaultJerk := DefaultJerk;
END_SET
END_PROPERTY

{attribute 'OPC.UA.DA.Property' := '1'}
{attribute 'monitoring':='call'}
//This value is used if commanded velocity is 0. Initvalue: Nc parameter manual velocity maximum
PROPERTY DefaultVelocity : LREAL
GET
DefaultVelocity := THIS^.fDefaultVelocity;
END_GET
SET
THIS^.fDefaultVelocity := DefaultVelocity;
END_SET
END_PROPERTY

{attribute 'OPC.UA.DA.Property' := '1'}
{attribute 'monitoring':='call'}
//Velocity override in % for all movement commands. (0 ≤ Override ≤ 100.0)
PROPERTY Override : LREAL
GET
Override := THIS^.fOverride;
END_GET
SET
//Syntax: OUT := LIMIT(Min, IN, Max) - Max is the upper bound, Min is the lower bound for the result. If the value IN exceeds the upper bound Max, LIMIT returns Max. If IN falls below Min, the result is Min.
THIS^.fOverride := LIMIT(0.0, Override, 100.0);
END_SET
END_PROPERTY

{attribute 'OPC.UA.DA.Property' := '1'}
{attribute 'monitoring':='call'}
PROPERTY SetAcceleration : LREAL
GET
SetAcceleration := THIS^.Axis.NcToPlc.SetAcc;
END_GET
END_PROPERTY

{attribute 'OPC.UA.DA.Property' := '1'}
{attribute 'monitoring':='call'}
PROPERTY SetPosition : LREAL
GET
SetPosition := THIS^.Axis.NcToPlc.SetPos;
END_GET
END_PROPERTY

{attribute 'OPC.UA.DA.Property' := '1'}
{attribute 'monitoring':='call'}
PROPERTY SetPosModulo : LREAL
GET
SetPosModulo := THIS^.Axis.NcToPlc.ModulosetPos;
END_GET
END_PROPERTY

{attribute 'OPC.UA.DA.Property' := '1'}
{attribute 'monitoring':='call'}
PROPERTY SetVelocity : LREAL
GET
SetVelocity := THIS^.Axis.NcToPlc.SetVelo;
END_GET
END_PROPERTY

{attribute 'OPC.UA.DA.Property' := '1'}
{attribute 'monitoring':='call'}
PROPERTY BufferEmpty : BOOL;
GET
VAR
	nCtsBusyCommands : UINT;
END_VAR
THIS^.Prepare();//Prepare time-critical information, if not already done

nCtsBusyCommands := nCtsBusyCommands + BOOL_TO_UINT(fbMoveRelative[0].Busy);
nCtsBusyCommands := nCtsBusyCommands + BOOL_TO_UINT(fbMoveRelative[1].Busy);
nCtsBusyCommands := nCtsBusyCommands + BOOL_TO_UINT(fbMoveAbsolute[0].Busy);
nCtsBusyCommands := nCtsBusyCommands + BOOL_TO_UINT(fbMoveAbsolute[1].Busy);
nCtsBusyCommands := nCtsBusyCommands + BOOL_TO_UINT(fbMoveVelocity[0].Busy);
nCtsBusyCommands := nCtsBusyCommands + BOOL_TO_UINT(fbMoveVelocity[1].Busy);
BufferEmpty := NOT bNewBufferCommadThisCycle AND NOT Axis.Status.CmdBuffered AND nCtsBusyCommands < 2;
END_GET
END_PROPERTY

{attribute 'OPC.UA.DA.Property' := '1'}
{attribute 'monitoring':='call'}
PROPERTY Coupled : BOOL
GET
THIS^.Prepare();//Prepare time-critical information, if not already done

Coupled := THIS^.Axis.Status.Coupled;
END_GET
END_PROPERTY

{attribute 'monitoring':='call'}
//operational and position control active
PROPERTY Enabled : BOOL
GET
THIS^.Prepare();//Prepare time-critical information, if not already done

(* StateDWord bit 20 - operational and position control active *)
Enabled :=  THIS^.Axis.Status.ControlLoopClosed;
END_GET
END_PROPERTY

{attribute 'OPC.UA.DA.Property' := '1'}
{attribute 'monitoring':='call'}
PROPERTY Feedback : I_CH_Feedback
GET
Feedback := THIS^.fbFeedback;
END_GET
END_PROPERTY

{attribute 'OPC.UA.DA.Property' := '1'}
{attribute 'monitoring':='call'}
PROPERTY LagDistance : LREAL
GET
LagDistance := THIS^.Axis.NcToPlc.PosDiff;
END_GET
END_PROPERTY

{attribute 'OPC.UA.DA.Property' := '1'}
{attribute 'monitoring':='call'}
PROPERTY MotionState : Tc2_MC2.MC_AxisStates
GET
THIS^.Prepare();//Prepare time-critical information, if not already done

MotionState := THIS^.Axis.Status.MotionState;
END_GET
END_PROPERTY

{attribute 'OPC.UA.DA.Property' := '1'}
{attribute 'monitoring':='call'}
PROPERTY Moving : BOOL
GET
THIS^.Prepare();//Prepare time-critical information, if not already done

Moving := THIS^.Axis.Status.Moving;
END_GET
END_PROPERTY

METHOD FB_init : BOOL
VAR_INPUT
	bInitRetains : BOOL; // if TRUE, the retain variables are initialized (warm start / cold start)
	bInCopyCode : BOOL;  // if TRUE, the instance afterwards gets moved into the copy code (online change)
END_VAR
//Do the following code once during start up and not during onlinechange
IF NOT bInCopyCode THEN 
	THIS^.fbFeedback.ActiveCommand 	:= TO_STRING(E_NcAxisCommands.None);	
END_IF
END_METHOD

METHOD Initialize : HRESULT
VAR_INST
	fbReadDriveAddress	: MC_ReadDriveAddress;
	fbReadParameterSet 	: MC_ReadParameterSet;
	
	stVarInfo : __SYSTEM.VAR_INFO;
END_VAR
VAR_INST
	//This error cannot be reset. Requires a reset cold
	{attribute 'hide'}	
	fbInitError : FB_TcAlarm;
END_VAR
IF NOT THIS^.bInitDone THEN
	THIS^.eActiveCommand 				:= E_NcAxisCommands.Initialize;
	THIS^.fbFeedback.ActiveCommand 		:= TO_STRING(THIS^.eActiveCommand);
	THIS^.fbFeedback.LastCommandAccepted:= TRUE;		


	
	// Check if link to NC is mapped
	IF NcParameterlist.ERROR_IF_NC_AXIS_IS_NOT_MAPPED AND NOT THIS^.Mapped THEN
		IF NOT fbInitError.bRaised THEN 
			//This error cannot be reset. Requires a reset cold
			fbInitError.CreateEx(	stEventEntry	:=TC_EVENTS.CHALET_NC_Events.VariableLinkMissing,
									ipSourceInfo 	:= THIS^.fbSourceInfo, 
									bWithConfirmation := FALSE);
			stVarInfo := __VARINFO(Axis);
			fbInitError.ipArguments.AddString(stVarInfo.Symbol);
			fbInitError.Raise(0);
		END_IF
		Initialize := E_FAIL;
		RETURN;
	END_IF

	
	// Check and wait until NC Task is in a valid running state
	IF NcParameterlist.ERROR_IF_NC_AXIS_IS_NOT_MAPPED AND THIS^.Axis.NcToPlc.AxisId = 0 THEN
		GetMostSignificant(Initialize, S_Pending);
		RETURN;
	END_IF
	
	
	// Get Drive Address on startup  	
	fbReadDriveAddress(
		Axis:= THIS^.Axis, 
		Execute:= NOT (fbReadDriveAddress.Busy OR fbReadDriveAddress.Done),
		DriveAddress=> THIS^.Axis.DriveAddress);
		
		
	// Read all axis parameter on startup
	fbReadParameterSet(
		Parameter:= stAxisParameterSet, 
		Axis:= THIS^.Axis, 
		Execute:= NOT (fbReadParameterSet.Busy OR fbReadParameterSet.Done), 
		ErrorID=> );
		
		
	// Store default values of parameterset in local variabels
	IF fbReadParameterSet.Done THEN
		fDefaultVelocity 		:= THIS^.stAxisParameterSet.fVeloFastManual;
		fDefaultAcceleration 	:= THIS^.stAxisParameterSet.fAcceleration;
		fDefaultDeceleration 	:= THIS^.stAxisParameterSet.fDeceleration;
		fDefaultJerk 			:= THIS^.stAxisParameterSet.fJerk;	
	END_IF
	
		
	// Set init done signal  
	THIS^.bInitDone := fbReadDriveAddress.Done AND fbReadParameterSet.Done AND Initialize = S_OK;
		
END_IF

THIS^.fbFeedback.HR := Initialize;
END_METHOD

{attribute 'monitoring':='call'}
PROPERTY Initialized : BOOL
GET
Initialized := THIS^.bInitDone;
END_GET
END_PROPERTY

(* 	Use this Methode to calculate time sensitive date once each cycle. Example: read analog input and convert before do get Signal propertie*)
METHOD PROTECTED Prepare : HRESULT
VAR
	bErrorCondition : BOOL;
END_VAR
VAR_INST
	{attribute 'hide'}	
	nLastUpdatedCycleCount : UDINT;
	{attribute 'hide'}	
	nOldErrorCode 		: UDINT;
	{attribute 'hide'}	
	fbAlarmNc			: FB_TcAlarm;
	{attribute 'hide'}
	fbAlarmInvalideIoData	: FB_TcAlarm;	
	{attribute 'hide'}
	fbAlarmDriveDeviceError	: FB_TcAlarm;	
	{attribute 'hide'}
	fbAlarmSoftLimitMinExceeded	: FB_TcAlarm;	
	{attribute 'hide'}
	fbAlarmSoftLimitMaxExceeded	: FB_TcAlarm;
END_VAR
//Check if this Cycle the dates are allready prepared. This is important for time sensitive informations.
IF nLastUpdatedCycleCount <> TwinCAT_SystemInfoVarList._TaskInfo[THIS^.TaskIndex].CycleCount THEN
	nLastUpdatedCycleCount := TwinCAT_SystemInfoVarList._TaskInfo[THIS^.TaskIndex].CycleCount ;

	
	// Refresh Axis Information 
	Axis.ReadStatus();
	
	
	
	//Write NC-Error(Axis.NcToPlc.ErrorCode) in TC3 Eventlogger
	bErrorCondition := NOT (THIS^.Axis.NcToPlc.ErrorCode = 0);
	IF (NOT bErrorCondition AND fbAlarmNc.bRaised) THEN
		//No error - Reset	
		fbAlarmNc.Clear(0,0);
		
	ELSIF (NOT bErrorCondition) THEN
		; //Nothing
		
	ELSIF (nOldErrorCode <> THIS^.Axis.NcToPlc.ErrorCode) THEN
		//New Error - Reset, Create and Raise
		fbAlarmNc.Clear(0,0);
		fbAlarmNc.Create(	eventClass		:= TC_EVENT_CLASSES.Tc3_NcErrorCodes, 
							nEventId		:= THIS^.Axis.NcToPlc.ErrorCode, 
							eSeverity		:= TcEventSeverity.Error, 
							ipSourceInfo 	:= THIS^.fbSourceInfo, 
							bWithConfirmation := FALSE);
		fbAlarmNc.ipArguments.Clear();
		fbAlarmNc.Raise(0);
	ELSE
		//Alarm is already active
		;
	END_IF
	nOldErrorCode := THIS^.Axis.NcToPlc.ErrorCode;
	
	
	
	//Write InvalideIoData(Axis.NcToPlc.StateDWord.30) in TC3 Eventlogger
	bErrorCondition := THIS^.Axis.NcToPlc.StateDWord.30;
	IF (NOT bErrorCondition AND fbAlarmInvalideIoData.bRaised) THEN
		//No error - Reset	
		fbAlarmInvalideIoData.Clear(0,0);
		
	ELSIF (NOT bErrorCondition) THEN
		; //Nothing
			
	ELSIF (bErrorCondition AND NOT fbAlarmInvalideIoData.bRaised) THEN
		//New Error - Create and Raise
		fbAlarmInvalideIoData.CreateEx(	
					stEventEntry:= TC_EVENTS.CHALET_NC_Events.IoDataInvalid,
					ipSourceInfo 	:= THIS^.fbSourceInfo, 
					bWithConfirmation := FALSE);
		fbAlarmInvalideIoData.ipArguments.Clear();
		fbAlarmInvalideIoData.Raise(0);
	ELSE
		//Alarm is already active
		;
	END_IF
	
	
	
	//Write DriveDeviceError(Axis.NcToPlc.StateDWord.28) in TC3 Eventlogger. Ignore if axis is disabled, to many errors in STO
	bErrorCondition := THIS^.Axis.NcToPlc.StateDWord.28 AND THIS^.Enabled;
	IF (NOT bErrorCondition AND fbAlarmDriveDeviceError.bRaised) THEN
		//No error - Reset	
		fbAlarmDriveDeviceError.Clear(0,0);
				
	ELSIF (NOT bErrorCondition) THEN
		; //Nothing
		
	ELSIF (bErrorCondition AND NOT fbAlarmDriveDeviceError.bRaised) THEN
		//New Error - Create and Raise
		fbAlarmDriveDeviceError.CreateEx(	
					stEventEntry:= TC_EVENTS.CHALET_NC_Events.DriveDeviceError,
					ipSourceInfo 	:= THIS^.fbSourceInfo, 
					bWithConfirmation := FALSE);
		fbAlarmDriveDeviceError.ipArguments.Clear();
		fbAlarmDriveDeviceError.Raise(0);
	ELSE
		//Alarm is already active
		;
	END_IF
	
	
	
	//Write SoftLimitMinExceeded(Axis.NcToPlc.StateDWord.26) in TC3 Eventlogger
	bErrorCondition := THIS^.Axis.NcToPlc.StateDWord.26;
	IF (NOT bErrorCondition AND fbAlarmSoftLimitMinExceeded.bRaised) THEN
		//No error - Reset	
		fbAlarmSoftLimitMinExceeded.Clear(0,0);		
		
	ELSIF (NOT bErrorCondition) THEN
		; //Nothing
	
	ELSIF (bErrorCondition AND NOT fbAlarmSoftLimitMinExceeded.bRaised) THEN
		//New Error - Create and Raise
		fbAlarmSoftLimitMinExceeded.CreateEx(	
					stEventEntry:= TC_EVENTS.CHALET_NC_Events.SoftLimitMinExceeded,
					ipSourceInfo 	:= THIS^.fbSourceInfo, 
					bWithConfirmation := FALSE);
		fbAlarmSoftLimitMinExceeded.ipArguments.Clear();
		fbAlarmSoftLimitMinExceeded.Raise(0);
	ELSE
		//Alarm is already active
		;
	END_IF
	
	
	
	//Write SoftLimitMaxExceeded(Axis.NcToPlc.StateDWord.27) in TC3 Eventlogger
	bErrorCondition := THIS^.Axis.NcToPlc.StateDWord.27;
	IF (NOT bErrorCondition AND fbAlarmSoftLimitMaxExceeded.bRaised) THEN
		//No error - Reset	
		fbAlarmSoftLimitMaxExceeded.Clear(0,0);
				
	ELSIF (NOT bErrorCondition) THEN
		; //Nothing
	
	ELSIF (bErrorCondition AND NOT fbAlarmSoftLimitMaxExceeded.bRaised) THEN
		//New Error - Create and Raise
		fbAlarmSoftLimitMaxExceeded.CreateEx(	
					stEventEntry:= TC_EVENTS.CHALET_NC_Events.SoftLimitMaxExceeded,
					ipSourceInfo 	:= THIS^.fbSourceInfo, 
					bWithConfirmation := FALSE);
		fbAlarmSoftLimitMaxExceeded.ipArguments.Clear();
		fbAlarmSoftLimitMaxExceeded.Raise(0);
	ELSE
		//Alarm is already active
		;
	END_IF
	
END_IF
END_METHOD

METHOD Update  : HRESULT
VAR
	//Gear
	{attribute 'hide'}
	fbGearMasterAxisRef  	: REFERENCE TO TC2_MC2.AXIS_REF; //Interface call in the Update methode to get this Referenz. Online-Change safe	
	
	//Multigear
	{attribute 'hide'}
	fbMultiGearMasterAxisRef1	: REFERENCE TO TC2_MC2.AXIS_REF; //Interface call in the Update methode to get this Referenz. Online-Change safe	
	{attribute 'hide'}
	fbMultiGearMasterAxisRef2	: REFERENCE TO TC2_MC2.AXIS_REF; //Interface call in the Update methode to get this Referenz. Online-Change safe	
	{attribute 'hide'}
	fbMultiGearMasterAxisRef3	: REFERENCE TO TC2_MC2.AXIS_REF; //Interface call in the Update methode to get this Referenz. Online-Change safe	
	{attribute 'hide'}
	fbMultiGearMasterAxisRef4	: REFERENCE TO TC2_MC2.AXIS_REF; //Interface call in the Update methode to get this Referenz. Online-Change safe	
END_VAR
// ********************** Do initialisation first ***********************************************
IF NOT THIS^.bInitDone THEN
	Update := THIS^.Initialize();
	RETURN;
END_IF

// ********************** Refresh Axis Information ***********************************************
THIS^.Prepare();//Prepare time-critical information, if not already done


// ********************** Set feedback depending on active command *******************************
CASE THIS^.eActiveCommand OF
	E_NcAxisCommands.None: 
		//Display if a NC Error is active during no command is active
		IF THIS^.Axis.Status.Error AND NOT fbFeedback.Error THEN 
			fbFeedback.ActiveCommand 	:= TO_STRING(E_NcAxisCommands.None);			
			fbFeedback.ErrorId 			:= THIS^.Axis.Status.ErrorID;
		END_IF
		
	E_NcAxisCommands.Initialize:
		fbFeedback.Busy 		:= NOT THIS^.bInitDone;
		fbFeedback.Done 		:= THIS^.bInitDone;
		fbFeedback.ErrorId 		:= 0;
		
	E_NcAxisCommands.Reset:
		fbFeedback.Busy 		:= fbReset.Busy;
		fbFeedback.Done 		:= fbReset.Done;
		fbFeedback.ErrorId 		:= fbReset.ErrorID;

	E_NcAxisCommands.PowerOn:
		fbFeedback.Busy 		:= fbPower.Busy;
		fbFeedback.Done 		:= fbPower.Status;
		fbFeedback.ErrorId 		:= fbPower.ErrorID;

	E_NcAxisCommands.PowerOff:
		fbFeedback.Busy 		:= fbPower.Busy;
		fbFeedback.Done 		:= THIS^.Axis.Status.Disabled;
		fbFeedback.ErrorId 		:= fbPower.ErrorID;
		
	E_NcAxisCommands.SetPosition:
		fbFeedback.Busy 		:= fbSetPosition.Busy;
		fbFeedback.Done 		:= fbSetPosition.Done;
		fbFeedback.ErrorId 		:= fbSetPosition.ErrorID;
		
	E_NcAxisCommands.Homing:
		fbFeedback.Busy 		:= fbHoming.Busy;
		fbFeedback.Done 		:= fbHoming.Done;
		fbFeedback.ErrorId 		:= fbHoming.ErrorID;
		
	E_NcAxisCommands.Stop: 
		fbFeedback.Busy 		:= fbStop.Busy;
		fbFeedback.Done 		:= (fbStop.Done OR NOT fbStop.Execute) AND NOT fbStop.Busy;
		fbFeedback.ErrorId 		:= fbStop.ErrorID;
		
		//FB_Stop: The Busy output becomes TRUE when the command is started with Execute and remains TRUE as long as the command is processed. If Busy becomes FALSE again, the function block is ready for a new job.
		//Attention: Busy remains TRUE as long as the axis is locked. The axis is only unlocked and Busy becomes FALSE when Execute is set to FALSE.
		IF fbStop.Done THEN
			fbStop.Execute := FALSE;
		END_IF
		
	E_NcAxisCommands.MoveVelocity:
		fbFeedback.Busy 		:= fbMoveVelocity[nActiveMoveVel].Busy;
		fbFeedback.Done 		:= fbMoveVelocity[nActiveMoveVel].InVelocity;
		fbFeedback.ErrorId 		:= fbMoveVelocity[nActiveMoveVel].ErrorID;

	E_NcAxisCommands.MoveRelative:
		fbFeedback.Busy 		:= fbMoveRelative[nActiveMoveRel].Busy;
		fbFeedback.Done 		:= fbMoveRelative[nActiveMoveRel].Done;
		fbFeedback.ErrorId 		:= fbMoveRelative[nActiveMoveRel].ErrorID;
	
	E_NcAxisCommands.MoveAbsolute:
		fbFeedback.Busy 		:= fbMoveAbsolute[nActiveMoveAbs].Busy;
		fbFeedback.Done 		:= fbMoveAbsolute[nActiveMoveAbs].Done;
		fbFeedback.ErrorId 		:= fbMoveAbsolute[nActiveMoveAbs].ErrorID;
			
	E_NcAxisCommands.GearIn:	
		fbFeedback.Busy 		:= fbGearIn.Busy;
		fbFeedback.Done 		:= fbGearIn.InGear;
		fbFeedback.ErrorId 		:= fbGearIn.ErrorID;
		
	E_NcAxisCommands.GearOut:
		fbFeedback.Busy 		:= fbGearOut.Busy;
		fbFeedback.Done 		:= fbGearOut.Done;
		fbFeedback.ErrorId 		:= fbGearOut.ErrorID;
			
	E_NcAxisCommands.MultiGearIn:
		//Wait for the GearOut to finish before GearIn
		THIS^.fbGearInMultiMaster.Enable := NOT THIS^.Axis.Status.Coupled;
		fbFeedback.Busy 		:= fbGearInMultiMaster.Busy;
		fbFeedback.Done 		:= fbGearInMultiMaster.InGear;
		fbFeedback.ErrorId 		:= fbGearInMultiMaster.ErrorID;
		
	ELSE//External command in subclass
		;
END_CASE


// **********************  Stop to execute commands on .done or .error ***************************
IF THIS^.fbFeedback.Done OR THIS^.fbFeedback.Error THEN
	eActiveCommand 				:= E_NcAxisCommands.None;
END_IF


// ******  Get master axis AXIS_REF for gear - Only call if interface to masteraxis is valide else dummy axis ******
IF THIS^.ipGearMasterAxis <> 0 THEN
	fbGearMasterAxisRef REF= THIS^.ipGearMasterAxis.getAxisRef;
ELSE
	fbGearMasterAxisRef REF= THIS^.fbDummyAxisRef;
END_IF
IF THIS^.ipMultiGearMasterAxis1 <> 0 THEN
	fbMultiGearMasterAxisRef1 REF= THIS^.ipMultiGearMasterAxis1.getAxisRef;
ELSE
	fbMultiGearMasterAxisRef1 REF= THIS^.fbDummyAxisRef;
END_IF
IF THIS^.ipMultiGearMasterAxis2 <> 0 THEN
	fbMultiGearMasterAxisRef2 REF= THIS^.ipMultiGearMasterAxis2.getAxisRef;
ELSE
	fbMultiGearMasterAxisRef2 REF= THIS^.fbDummyAxisRef;
END_IF
IF THIS^.ipMultiGearMasterAxis3 <> 0 THEN
	fbMultiGearMasterAxisRef3 REF= THIS^.ipMultiGearMasterAxis3.getAxisRef;
ELSE
	fbMultiGearMasterAxisRef3 REF= THIS^.fbDummyAxisRef;
END_IF
IF THIS^.ipMultiGearMasterAxis4 <> 0 THEN
	fbMultiGearMasterAxisRef4 REF= THIS^.ipMultiGearMasterAxis4.getAxisRef;
ELSE
	fbMultiGearMasterAxisRef4 REF= THIS^.fbDummyAxisRef;
END_IF


// **********************  Cyclic calls  *********************************************************
fbPower(Axis 			:= THIS^.Axis, 
		Override 		:= THIS^.fOverride,
		Enable_Positive := NOT THIS^.bLockPositiveDirection,
		Enable_Negative := NOT THIS^.bLockNegativeDirection);
fbStop(Axis := THIS^.Axis);
fbReset(Axis := THIS^.Axis);
fbHoming(	Axis := THIS^.Axis);
fbGearOut(Slave := THIS^.Axis);
fbSetPosition(Axis := THIS^.Axis);
fbMoveRelative[0](Axis := THIS^.Axis); 
fbMoveRelative[1](Axis := THIS^.Axis);
fbMoveAbsolute[0](Axis := THIS^.Axis); 
fbMoveAbsolute[1](Axis := THIS^.Axis);
fbMoveVelocity[0](Axis := THIS^.Axis); 
fbMoveVelocity[1](Axis := THIS^.Axis);
fbGearIn(	Master 	:= fbGearMasterAxisRef, 
			Slave 	:= THIS^.Axis);
fbGearInMultiMaster(	Master1		:=fbMultiGearMasterAxisRef1, 
						Master2		:=fbMultiGearMasterAxisRef2,
					 	Master3		:=fbMultiGearMasterAxisRef3, 
						Master4		:=fbMultiGearMasterAxisRef4, 
						Slave		:=THIS^.Axis);
						
						
// ********************** Reset all Execution flags **********************************************
fbGearinMultiMaster.Enable := FALSE;
fbStop.Execute := FALSE;
fbReset.Execute := FALSE;
fbHoming.Execute := FALSE;
fbGearOut.Execute := FALSE;
fbSetPosition.Execute := FALSE;
fbGearIn.Execute := FALSE;
fbMoveRelative[0].Execute := FALSE;
fbMoveRelative[1].Execute := FALSE;
fbMoveAbsolute[0].Execute := FALSE;
fbMoveAbsolute[1].Execute := FALSE;
fbMoveVelocity[0].Execute := FALSE;
fbMoveVelocity[1].Execute := FALSE;


// This flag is processed in the PLC cycle when a buffered motion command is requested via method
THIS^.bNewBufferCommadThisCycle := FALSE;

// ****************Get the acive instance. Stay at the last active.********************************
IF fbMoveVelocity[0].Active THEN
	nActiveMoveVel := 0;
ELSIF fbMoveVelocity[1].Active THEN
	nActiveMoveVel := 1;
END_IF

IF fbMoveRelative[0].Active THEN
	nActiveMoveRel := 0;
ELSIF fbMoveRelative[1].Active THEN
	nActiveMoveRel := 1;
END_IF

IF fbMoveAbsolute[0].Active THEN
	nActiveMoveAbs := 0;
ELSIF fbMoveAbsolute[1].Active THEN
	nActiveMoveAbs := 1;
END_IF

//Return
Update := THIS^.fbFeedback.HR;
END_METHOD

END_FUNCTION_BLOCK

// COMPONENTs/Optional/Adapter AXIS_REF/FB_Adapter_AXIS_REF
FUNCTION_BLOCK FB_Adapter_AXIS_REF EXTENDS FB_CH_Object IMPLEMENTS I_Adapter_AXIS_REF
VAR
	Axis : Tc2_Mc2.AXIS_REF;
END_VAR

PROPERTY getAxisRef : REFERENCE TO Tc2_MC2.AXIS_REF
GET
getAxisRef REF= THIS^.Axis;
END_GET
END_PROPERTY

END_FUNCTION_BLOCK

// COMPONENTs/Optional/Adapter AXIS_REF/I_Adapter_AXIS_REF
INTERFACE I_Adapter_AXIS_REF

PROPERTY getAxisRef : REFERENCE TO Tc2_MC2.AXIS_REF
GET
END_GET
END_PROPERTY

END_INTERFACE

// COMPONENTs/Main FB/I_NcAxis_PLC
INTERFACE I_NcAxis_PLC EXTENDS I_AxisStatus, I_Adapter_AXIS_REF

{attribute 'TcRpcEnable':='1'} //call methode via OPC-UA connection
(*! 
<summary>
	Establish an axis coupling to a single master axis.
	<preliminary>
		Both axis must be in standstill to apply the coupling.
		In-motion coupling of the FB is not supported by this method.
	</preliminary>
</summary>
<description>
	The coupling is performed based on a <b>velocity</b> ratio.
	As reference the master axis <b>command</b> value is used.
	There is <b>no automatic phase compensation</b> applied.
	
	<h3> Missing features </h3>
	<ul> 
		<li> - </li>
		<li> - </li>
	</ul>
</description> 
*)

METHOD PUBLIC GearIn  : I_CH_Feedback (*! Interface to the execution feedback *)
VAR_INPUT
	(*! Interface to a master axis *)
	ipMasterAxisAdapter : I_Adapter_AXIS_REF;

	(*! Gear ratio Numerator*)
	fRatioNumerator: LREAL;
	
	(*! Gear ratio Denominator*)
	nRatioDenominator: UINT;
	
	(*! Use the default dynamics if input=0.
	The default dynamics can be read and written via property and is initialized with the default values in the NC parameter list. *)
	fAcceleration	: LREAL;
	
	(*! Use the default dynamics if input=0. 
	The default dynamics can be read and written via property and is initialized with the default values in the NC parameter list. *)
	fDeceleration	: LREAL;
	
	(*! Use the default dynamics if input=0. 
	The default dynamics can be read and written via property and is initialized with the default values in the NC parameter list. *)
	fJerk			: LREAL;
END_VAR
END_METHOD

{attribute 'TcRpcEnable':='1'} 
(*WARNING
No standstill of the axis due to decoupling
When a slave axis is uncoupled during the movement, it is not stopped automatically but reaches a constant velocity at which it continues to travel infinitely.
You can stop the axis with the function blocks MC_Halt or MC_Stop.*)
METHOD GearOut  : I_CH_Feedback
END_METHOD

{attribute 'TcRpcEnable':='1'} 
(*The parameterization of the home command takes place in the NC! To do this, set the parameters in:
- NC-Axis(Parameters) Homing speed
- NC-Axis>Encoder(Parameters) Homing mode
	Reference Mode: "Homing Sensor Only"
	Homing Sensor Source "Digital Input x" 
		Link Input to NC-Axis>Drive>Inputs>nState8.x
*)
(*Homing refers to an axis initialization run during which the correct actual position is determined by means of a reference signal. This can be NC-guided, as default described here:
  - The axis is at a random position.
  - The axis moves in the parameterized direction and searches for the reference switch (referencing cam/calibration cam).
  - The axis reverses as soon as the referencing cam is detected.
  - The axis moves away from the referencing cam and detects the falling edge of the cam signal.
  - The axis continues to move and searches for the sync pulse (latch signal or zero pulse of the encoder).
  - The reference position is set and the axis stops. The standstill position of the axis deviates slightly from the reference position.*)
METHOD Homing  : I_CH_Feedback
VAR_INPUT
	(*Absolute reference position to which the axis is set after homing*)
	fPosition		: LREAL;
END_VAR
END_METHOD

{attribute 'monitoring':='call'}
//Disable the feed in one direction.
PROPERTY LockNegativeDirection : BOOL
GET
END_GET
SET
END_SET
END_PROPERTY

{attribute 'monitoring':='call'}
//Disable the feed in one direction.
PROPERTY LockPositiveDirection : BOOL
GET
END_GET
SET
END_SET
END_PROPERTY

{attribute 'TcRpcEnable':='1'} 
METHOD MoveAbsolute  : I_CH_Feedback
VAR_INPUT
	fPosition		: LREAL;
	
	(* Use the default dynamics if input=0. 
	The default dynamics can be read and written via property and is initialized with the default values in the NC parameter list. *)
	fVelocity		: LREAL;
	
	(* Use the default dynamics if input=0. 
	The default dynamics can be read and written via property and is initialized with the default values in the NC parameter list. *)
	fAcceleration	: LREAL;
	
	(* Use the default dynamics if input=0. 
	The default dynamics can be read and written via property and is initialized with the default values in the NC parameter list. *)
	fDeceleration	: LREAL;
	
	(* Use the default dynamics if input=0. 
	The default dynamics can be read and written via property and is initialized with the default values in the NC parameter list. *)
	fJerk			: LREAL;
	
	(* Input=0 = MC_Aborting   
	BufferModes:
		-MC_Aborting: Default mode without buffering. The command is executed immediately and interrupts any other command that may be running.
		-MC_Buffered: The command is executed once no other command is running on the axis. The previous movement continues until it has stopped. The following command is started from standstill.
		-MC_BlendingLow: The command is executed once no other command is running on the axis. In contrast to Buffered the axis does not stop at the previous target, but passes through this position with the lower velocity of two commands.
		-MC_BlendingHigh The command is executed once no other command is running on the axis. In contrast to Buffered the axis does not stop at the previous target, but passes through this position with the higher velocity of two commands.
		-MC_BlendingNext: The command is executed once no other command is running on the axis. In contrast to Buffered the axis does not stop at the previous target, but passes through this position with the velocity of the last command.
		-MC_BlendingPrevious: The command is executed once no other command is running on the axis. In contrast to Buffered the axis does not stop at the previous target, but passes through this position with the velocity of the first command. *)
	eBufferMode   : Tc2_MC2.MC_BufferMode;
END_VAR
END_METHOD

{attribute 'TcRpcEnable':='1'} 
METHOD MoveRelative  : I_CH_Feedback
VAR_INPUT
	fDistance		: LREAL;
	
	(* Use the default dynamics if input=0. 
	The default dynamics can be read and written via property and is initialized with the default values in the NC parameter list. *)
	fVelocity		: LREAL;
	
	(* Use the default dynamics if input=0. 
	The default dynamics can be read and written via property and is initialized with the default values in the NC parameter list. *)
	fAcceleration	: LREAL;
	
	(* Use the default dynamics if input=0. 
	The default dynamics can be read and written via property and is initialized with the default values in the NC parameter list. *)
	fDeceleration	: LREAL;
	
	(* Use the default dynamics if input=0. 
	The default dynamics can be read and written via property and is initialized with the default values in the NC parameter list. *)
	fJerk			: LREAL;
	
	(* Input=0 = MC_Aborting   
	BufferModes:
		-MC_Aborting: Default mode without buffering. The command is executed immediately and interrupts any other command that may be running.
		-MC_Buffered: The command is executed once no other command is running on the axis. The previous movement continues until it has stopped. The following command is started from standstill.
		-MC_BlendingLow: The command is executed once no other command is running on the axis. In contrast to Buffered the axis does not stop at the previous target, but passes through this position with the lower velocity of two commands.
		-MC_BlendingHigh The command is executed once no other command is running on the axis. In contrast to Buffered the axis does not stop at the previous target, but passes through this position with the higher velocity of two commands.
		-MC_BlendingNext: The command is executed once no other command is running on the axis. In contrast to Buffered the axis does not stop at the previous target, but passes through this position with the velocity of the last command.
		-MC_BlendingPrevious: The command is executed once no other command is running on the axis. In contrast to Buffered the axis does not stop at the previous target, but passes through this position with the velocity of the first command. *)
	eBufferMode   : Tc2_MC2.MC_BufferMode;
END_VAR
END_METHOD

{attribute 'TcRpcEnable':='1'} 
METHOD MoveVelocity  : I_CH_Feedback
VAR_INPUT
	(* Use the default dynamics if input=0. 
	The default dynamics can be read and written via property and is initialized with the default values in the NC parameter list. *)
	fVelocity		: LREAL;
	
	(* Use the default dynamics if input=0. 
	The default dynamics can be read and written via property and is initialized with the default values in the NC parameter list. *)
	fAcceleration	: LREAL;
	
	(* Use the default dynamics if input=0. 
	The default dynamics can be read and written via property and is initialized with the default values in the NC parameter list. *)
	fDeceleration	: LREAL;
	
	(* Use the default dynamics if input=0. 
	The default dynamics can be read and written via property and is initialized with the default values in the NC parameter list. *)
	fJerk			: LREAL;
	
	(* If input=1, then direction is positive. 
	Positive OR negative direction of travel (TYPE: Tc2_MC2.MC_Direction) *)
	eDirection: Tc2_MC2.MC_Direction;
	
	(* Input=0 = MC_Aborting   
	BufferModes:
		-MC_Aborting: Default mode without buffering. The command is executed immediately and interrupts any other command that may be running.
		-MC_Buffered: The command is executed once no other command is running on the axis. The previous movement continues until it has stopped. The following command is started from standstill.
		-MC_BlendingLow: The command is executed once no other command is running on the axis. In contrast to Buffered the axis does not stop at the previous target, but passes through this position with the lower velocity of two commands.
		-MC_BlendingHigh The command is executed once no other command is running on the axis. In contrast to Buffered the axis does not stop at the previous target, but passes through this position with the higher velocity of two commands.
		-MC_BlendingNext: The command is executed once no other command is running on the axis. In contrast to Buffered the axis does not stop at the previous target, but passes through this position with the velocity of the last command.
		-MC_BlendingPrevious: The command is executed once no other command is running on the axis. In contrast to Buffered the axis does not stop at the previous target, but passes through this position with the velocity of the first command. *)
	eBufferMode   : Tc2_MC2.MC_BufferMode;
END_VAR
END_METHOD

{attribute 'TcRpcEnable':='1'} 
METHOD MultiGearIn : I_CH_Feedback
VAR_INPUT
	(* Interface to an master axis *)
	ipMasterAxisAdapter : I_Adapter_AXIS_REF;
	
	(* Gear ratio Numerator*)
	fRatioNumerator: LREAL;
	(* Gear ratio Denominator*)
	nRatioDenominator: UINT;
	
	(* Use the default dynamics if input=0. 
	The default dynamics can be read and written via property and is initialized with the default values in the NC parameter list. *)
	fAcceleration	: LREAL;
	
	(* Use the default dynamics if input=0. 
	The default dynamics can be read and written via property and is initialized with the default values in the NC parameter list. *)
	fDeceleration	: LREAL;
	
	(* Use the default dynamics if input=0. 
	The default dynamics can be read and written via property and is initialized with the default values in the NC parameter list. *)
	fJerk			: LREAL;
END_VAR
END_METHOD

{attribute 'TcRpcEnable':='1'} 
METHOD PowerOff  : I_CH_Feedback
END_METHOD

{attribute 'TcRpcEnable':='1'} 
METHOD PowerOn : I_CH_Feedback
END_METHOD

METHOD Reset : I_CH_Feedback
VAR_INPUT
END_VAR
END_METHOD

{attribute 'TcRpcEnable':='1'} 
METHOD SetActPosition : I_CH_Feedback
VAR_INPUT
	fPosition: LREAL;
END_VAR
END_METHOD

{attribute 'TcRpcEnable':='1'} 
METHOD Stop : I_CH_Feedback
VAR_INPUT
	(* Use the default dynamics if input=0. 
	The default dynamics can be read and written via property and is initialized with the default values in the NC parameter list. *)
	fDeceleration: LREAL;
	
	(* Use the default dynamics if input=0. 
	The default dynamics can be read and written via property and is initialized with the default values in the NC parameter list. *)
	fJerk: LREAL;
END_VAR
END_METHOD

{attribute 'OPC.UA.DA.Property' := '1'}
{attribute 'monitoring':='call'}
PROPERTY ActAcceleration : LREAL
GET
END_GET
END_PROPERTY

{attribute 'OPC.UA.DA.Property' := '1'}
{attribute 'monitoring':='call'}
PROPERTY ActPosition : LREAL
GET
END_GET
END_PROPERTY

{attribute 'OPC.UA.DA.Property' := '1'}
{attribute 'monitoring':='call'}
PROPERTY ActPosModulo : LREAL
GET
END_GET
END_PROPERTY

{attribute 'OPC.UA.DA.Property' := '1'}
{attribute 'monitoring':='call'}
PROPERTY ActVelocity : LREAL
GET
END_GET
END_PROPERTY

{attribute 'OPC.UA.DA.Property' := '1'}
{attribute 'monitoring':='call'}
PROPERTY DefaultAcceleration : LREAL
GET
END_GET
SET
END_SET
END_PROPERTY

{attribute 'OPC.UA.DA.Property' := '1'}
{attribute 'monitoring':='call'}
PROPERTY DefaultDeceleration : LREAL
GET
END_GET
SET
END_SET
END_PROPERTY

{attribute 'OPC.UA.DA.Property' := '1'}
{attribute 'monitoring':='call'}
PROPERTY DefaultJerk : LREAL
GET
END_GET
SET
END_SET
END_PROPERTY

{attribute 'OPC.UA.DA.Property' := '1'}
{attribute 'monitoring':='call'}
//This value is used if commanded velocity is 0. Initvalue: Nc parameter manual velocity maximum
PROPERTY DefaultVelocity : LREAL
GET
END_GET
SET
END_SET
END_PROPERTY

{attribute 'OPC.UA.DA.Property' := '1'}
{attribute 'monitoring':='call'}
//Velocity override in % for all movement commands. (0 ≤ Override ≤ 100.0)
PROPERTY Override : LREAL
GET
END_GET
SET
END_SET
END_PROPERTY

{attribute 'OPC.UA.DA.Property' := '1'}
{attribute 'monitoring':='call'}
PROPERTY BufferEmpty : BOOL;
GET
END_GET
END_PROPERTY

{attribute 'OPC.UA.DA.Property' := '1'}
{attribute 'monitoring':='call'}
PROPERTY NcAxisType : Tc2_MC2.E_NcAxisType
GET
END_GET
END_PROPERTY

{attribute 'OPC.UA.DA.Property' := '1'}
{attribute 'monitoring':='call'}
PROPERTY NcDriveType : Tc2_MC2.E_NcDriveType
GET
END_GET
END_PROPERTY

METHOD Initialize : HRESULT
END_METHOD

METHOD Update   : HRESULT
VAR_INPUT
END_VAR
END_METHOD

END_INTERFACE

// COMPONENTs/Main FB/I_AxisStatus
INTERFACE I_AxisStatus

{attribute 'OPC.UA.DA.Property' := '1'}
{attribute 'monitoring':='call'}
//Velocity override in % for all movement commands. (0 ≤ Override ≤ 100.0)
PROPERTY Override : LREAL
GET
END_GET
END_PROPERTY

{attribute 'OPC.UA.DA.Property' := '1'}
{attribute 'monitoring':='call'}
PROPERTY SetAcceleration : LREAL
GET
END_GET
END_PROPERTY

{attribute 'OPC.UA.DA.Property' := '1'}
{attribute 'monitoring':='call'}
PROPERTY SetPosition : LREAL
GET
END_GET
END_PROPERTY

{attribute 'OPC.UA.DA.Property' := '1'}
{attribute 'monitoring':='call'}
PROPERTY SetPosModulo : LREAL
GET
END_GET
END_PROPERTY

{attribute 'OPC.UA.DA.Property' := '1'}
{attribute 'monitoring':='call'}
PROPERTY SetVelocity : LREAL
GET
END_GET
END_PROPERTY

{attribute 'monitoring':='call'}
//operational and position control active
PROPERTY Enabled : BOOL
GET
END_GET
END_PROPERTY

{attribute 'OPC.UA.DA.Property' := '1'}
{attribute 'monitoring':='call'}
PROPERTY LagDistance : LREAL
GET
END_GET
END_PROPERTY

{attribute 'monitoring':='call'}
//Disable the feed in one direction.
PROPERTY LockNegativeDirection : BOOL
GET
END_GET
END_PROPERTY

{attribute 'monitoring':='call'}
//Disable the feed in one direction.
PROPERTY LockPositiveDirection : BOOL
GET
END_GET
END_PROPERTY

{attribute 'monitoring':='call'}
PROPERTY Mapped : BOOL
GET
END_GET
END_PROPERTY

{attribute 'OPC.UA.DA.Property' := '1'}
{attribute 'monitoring':='call'}
PROPERTY MotionState : Tc2_MC2.MC_AxisStates
GET
END_GET
END_PROPERTY

{attribute 'monitoring':='call'}
PROPERTY Feedback : I_CH_Feedback
GET
END_GET
END_PROPERTY

{attribute 'monitoring':='call'}
PROPERTY Initialized : BOOL
GET
END_GET
END_PROPERTY

END_INTERFACE

// COMPONENTs/Main FB/I_NcAxis_HMI
INTERFACE I_NcAxis_HMI EXTENDS I_AxisStatus

PROPERTY Coupled : BOOL
GET
END_GET
END_PROPERTY

{attribute 'monitoring':='call'}
PROPERTY LUID : STRING  //Locally unique identifier
GET
END_GET
END_PROPERTY

PROPERTY Moving : BOOL
GET
END_GET
END_PROPERTY

{attribute 'OPC.UA.DA.Property' := '1'}
{attribute 'monitoring':='call'}
PROPERTY NcAxisName : String(31)
GET
END_GET
END_PROPERTY

END_INTERFACE

// COMPONENTs/Optional/Feedback/FB_NcFeedback
{attribute 'no_explicit_call' := 'Do not call the body - Stick to OOP'}
//In addition to the normal FB_Feedback object on the CHALET-Base Library, 
//this function block also checks whether the set ErrorID has been defined 
//in the NC event list and retrieves the translation from there.
FUNCTION_BLOCK FB_NcFeedback EXTENDS CHALET_BaseComponents.FB_CH_Feedback
VAR

END_VAR

METHOD PROTECTED UpdateEventlogger : BOOL
VAR
	nHR : DWORD;
END_VAR
IF THIS^.ipSourceInfo = 0 THEN
	//No TC3_Eventlogger alarm if interface is empty
	RETURN;
END_IF


//New error, raise alarm
IF (THIS^.ErrorId <> THIS^.nOldErrorId) AND THIS^.Error THEN
	THIS^.fbAlarm.Clear(0,0);
	THIS^.fbAlarm.CreateEx(stEventEntry := TC_EVENTS.CHALET_Base_Events.FeedbackErrorCmd, ipSourceInfo := THIS^.ipSourceInfo, bWithConfirmation:= FALSE);
	//Error in feedback command {0} error id {1}
	
	//Convert to DWORD
	nHR := TO_DWORD(THIS^.HR);
	
	//Try to get some more details about error id
	IF THIS^.HR = E_FAIL THEN
		THIS^.fbAlarm.ipArguments.Clear().AddStringByValue(THIS^.ActiveCommand).AddStringByValue('E_FAIL');
		
	ELSIF ((nHR AND 16#FFFF_FF00) = 16#9811_0000) THEN
		THIS^.fbAlarm.ipArguments.Clear().AddStringByValue(THIS^.ActiveCommand).AddUDInt(THIS^.ErrorId).AddEventReferenceIdGuid(nEventId := THIS^.ErrorId, EventClass := TC_EVENT_CLASSES.TcSystemEventClass);
		;//Global error codes
			
	ELSIF ((nHR AND 16#FFFF_FF00) = 16#9811_0500) THEN
		THIS^.fbAlarm.ipArguments.Clear().AddStringByValue(THIS^.ActiveCommand).AddUDInt(THIS^.ErrorId).AddEventReferenceIdGuid(nEventId := THIS^.ErrorId, EventClass := TC_EVENT_CLASSES.TcRouterEventClass);
		;//Router error codes
			
	ELSIF ((nHR AND 16#FFFF_FF00) = 16#9811_0700) THEN
		THIS^.fbAlarm.ipArguments.Clear().AddStringByValue(THIS^.ActiveCommand).AddUDInt(THIS^.ErrorId).AddEventReferenceIdGuid(nEventId := THIS^.ErrorId, EventClass := TC_EVENT_CLASSES.TcGeneralAdsEventClass);
		;//General ADS errors
			
	ELSIF ((nHR AND 16#FFFF_FF00) = 16#9811_1000) THEN
		THIS^.fbAlarm.ipArguments.Clear().AddStringByValue(THIS^.ActiveCommand).AddUDInt(THIS^.ErrorId).AddEventReferenceIdGuid(nEventId := THIS^.ErrorId, EventClass := TC_EVENT_CLASSES.TcRTimeEventClass);
		;//RTime error codes
	
	//NC errors are in range HEX 4000-4C50 or 8100-8167	
	ELSIF (THIS^.ErrorId >= 16#4000 AND THIS^.ErrorId <= 16#4C50) OR (THIS^.ErrorId >= 16#8100 AND THIS^.ErrorId <= 16#8167) THEN
		THIS^.fbAlarm.ipArguments.Clear().AddStringByValue(THIS^.ActiveCommand).AddUDInt(THIS^.ErrorId).AddEventReferenceIdGuid(nEventId := THIS^.ErrorId, EventClass := TC_EVENT_CLASSES.Tc3_NcErrorCodes);
		;//NC Error
	
	ELSE
		THIS^.fbAlarm.ipArguments.Clear().AddStringByValue(THIS^.ActiveCommand).AddUDInt(THIS^.ErrorId);
	END_IF
	
	THIS^.fbAlarm.Raise(0);

	
//Busy, raise info
ELSIF (THIS^.Busy <> THIS^.bOldBusy) AND THIS^.Busy AND BaseParameterlist.B_WRITE_INFO_FEEDBACK_BUSY THEN
	THIS^.fbAlarm.Clear(0,0);
	THIS^.fbAlarm.CreateEx(stEventEntry := TC_EVENTS.CHALET_Base_Events.FeedbackBusy, ipSourceInfo := THIS^.ipSourceInfo, bWithConfirmation:= FALSE);
	THIS^.fbAlarm.ipArguments.Clear().AddStringByValue(THIS^.ActiveCommand);
	THIS^.fbAlarm.Raise(0);
	
//No error, clear alarm	
ELSIF NOT THIS^.Error AND NOT (THIS^.Busy AND BaseParameterlist.B_WRITE_INFO_FEEDBACK_BUSY) THEN
	THIS^.fbAlarm.Clear(0,0);
END_IF

THIS^.nOldErrorId 	:= THIS^.ErrorId;
THIS^.bOldBusy 		:= THIS^.Busy;
END_METHOD

END_FUNCTION_BLOCK

// COMPONENTs/Optional/Reset/FB_Reset_NC_Sercos_CANopen
{attribute 'hide_all_locals'}
FUNCTION_BLOCK FB_Reset_NC_Sercos_CANopen
VAR_INPUT
    Execute : BOOL;
END_VAR
VAR_OUTPUT
    Done    : BOOL;
    Busy    : BOOL;
    Error   : BOOL;
    ErrorID : UDINT;
END_VAR
VAR_IN_OUT
    Axis 	: AXIS_REF;
END_VAR
VAR 
	nSeq 				: UDINT :=0;
	nErrorID 			: UDINT;
	fbSoEReset			: TC2_MC2_DRIVE.FB_SoEReset;
	fbAxisReset			: Tc2_MC2.MC_Reset;
	fbTriggerExecute	: R_TRIG;
END_VAR

fbTriggerExecute(CLK:= THIS^.Execute);
IF fbTriggerExecute.Q THEN
	THIS^.Done			:=FALSE;
	THIS^.Busy			:=TRUE;
	THIS^.Error			:=FALSE;
	nSeq 				:= 1;
END_IF

IF NOT (THIS^.Busy OR THIS^.Execute) THEN
	fbSoEReset.Execute	:=FALSE;
	fbAxisReset.Execute	:=FALSE;
	THIS^.Done			:=FALSE;
	THIS^.Busy			:=FALSE;
	THIS^.Error			:=FALSE;
	THIS^.ErrorID 		:= 0;
	nSeq 				:= 0;
END_IF

CASE nSeq OF
	0: // ************************ wait for commands  ***********************************
		
	1:	// **********************  Reset Safety  *****************************************

		(* ToDo Reset Safety *)	
		(* ToDo Reset Safety *)	
		(* ToDo Reset Safety *)	
		(* ToDo Reset Safety *)	
		(* ToDo Reset Safety *)	
		(* ToDo Reset Safety *)	
		
		nSeq := 10;	 
		
	10:	// **********************  Check if Sercos reset is recuired *****************************************
		//If Sercos Axis and Sercos reset recuired, do a sercos reset first. Else do normal reset
		IF (THIS^.Axis.DriveAddress.NcDriveType = NcDriveType_Sercos) AND (THIS^.Axis.Status.ErrorID >=17408)AND (THIS^.Axis.Status.ErrorID <=18005) THEN
			fbSoEReset.Execute	:=TRUE;
			nSeq := 20;	 			
		ELSE
			fbAxisReset.Execute := TRUE;
			nSeq := 30;
		END_IF	

	20:	// *********************  Wait for Sercos Reset done ************************************************************	
		IF fbSoEReset.Error THEN
			IF (fbSoEReset.AdsErrId <> 0) THEN
				nErrorID := fbSoEReset.AdsErrId;
			ELSE
				nErrorID := fbSoEReset.SercosErrId;
			END_IF
			fbAxisReset.Execute := TRUE;
			//goto error seq
			nSeq := 10000+nSeq; 
		ELSIF NOT fbSoEReset.Busy THEN
			fbSoEReset.Execute	:=FALSE;
			fbAxisReset.Execute := TRUE;
			nSeq := 30;
		END_IF				
			
	30:	// **********************  Wait for NC reset done *****************************************
		IF fbAxisReset.Error THEN
			nErrorID := fbAxisReset.ErrorID;
			fbAxisReset.Execute:=FALSE;
			//goto error seq
			nSeq := 10000+nSeq; 
		ELSIF fbAxisReset.Done THEN
			fbAxisReset.Execute:=FALSE;
			nSeq := 100;
		END_IF	
		
	100: // ********************** reset done  *****************************************************
		THIS^.Done		:=TRUE;
		THIS^.Busy		:=FALSE;
		THIS^.Error		:=FALSE;
		
	10000..20000: // ************  display error ************************************************************
		THIS^.Done		:=FALSE;
		THIS^.Busy		:=FALSE;
		THIS^.Error		:=TRUE;
		THIS^.ErrorID	:=nErrorID;		
END_CASE

// **********************  Cyclic calls  ************************************************************
fbAxisReset(Axis := THIS^.Axis);		
fbSoEReset(Axis:= THIS^.Axis);

END_FUNCTION_BLOCK

// COMPONENTs/Optional/SetActPosition/FB_SetPosition_Beckhoff
//{attribute 'hide_all_locals'}
(*This FB reads out where the position offset is to be saved (NC/Drive/Encoder) and also stores
 it there. Works for ELM72xx, EL72xx, Ax8xxx and Ax5xxx*)
FUNCTION_BLOCK FB_SetPosition_Beckhoff
VAR_INPUT
    Execute  : BOOL;
    Position : LREAL; 
    Mode     : BOOL; // RELATIVE=True, ABSOLUTE=False (Default)
    //Options  : ST_SetPositionOptions; // only Feedback1 is supportet
END_VAR

VAR_OUTPUT
    Done    : BOOL;
    Busy    : BOOL;
    Error   : BOOL;
    ErrorID : UDINT;
	
	bStoredInNc : BOOL;
	bStoredInDrive : BOOL;
	bStoredInEncoder : BOOL;
END_VAR

VAR_IN_OUT
    Axis 	: AXIS_REF;
END_VAR

VAR 
	fPosition 			: LREAL;
	bMode     			: BOOL; // RELATIVE=True, ABSOLUTE=False (Default)
	nSeq 				: UDINT :=0;
	fbTriggerExecute	: R_TRIG;
	
	fbReadDriveType 	: FB_ReadDriveInfo;
	stDriveInfo 		: ST_DriveInfo;
	
	fbReadDriveAddress 	: MC_ReadDriveAddress;
	fbSetPosNC 			: MC_SetPosition;

	fbCoERead 			: FB_CoERead;
	fbSoERead 			: FB_SoERead;

	fbSetPositionOffset	: FB_SetPositionOffset;
	fbDeletePositionOffset : FB_DeletePositionOffset;
	bSetOffsetInNC		 : BOOL;
	
	eReadFromCoe :UINT := 99;
	eReadFromSoe :UINT := 99;
END_VAR

fbTriggerExecute(CLK:= THIS^.Execute);
//Reset on positive execution edge
IF fbTriggerExecute.Q THEN
	THIS^.Done	:= FALSE;
	THIS^.Busy	:= TRUE;
	THIS^.Error	:= FALSE;
	nSeq		:= 1;
	bMode 		:= Mode;
	fPosition 	:= Position;
END_IF

IF NOT (THIS^.Busy OR THIS^.Execute) THEN
	THIS^.Done			:=FALSE;
	THIS^.Busy			:=FALSE;
	THIS^.Error			:=FALSE;
	THIS^.ErrorID 		:= 0;
	nSeq				:= 0;
	bStoredInNc := FALSE;
	bStoredInDrive := FALSE;
	bStoredInEncoder := FALSE;	
END_IF

CASE nSeq OF
	
	0: //Nothing
		RETURN;
	
	1: //Init
		fbReadDriveType.Execute := FALSE;
		fbCoERead.Execute		:= FALSE; 
		fbSetPosNC.Execute		:= FALSE; 
		bSetOffsetInNC			:= FALSE; 
		fbReadDriveAddress.Execute := FALSE;
		fbSetPositionOffset.Execute	:= FALSE; 
		fbDeletePositionOffset.Execute	:= FALSE; 
		nSeq := 10;

	10: //Read drive type
		fbReadDriveType.Execute  := TRUE;
		nSeq := 11;
		
	11:	//Read drive type
		IF fbReadDriveType.ErrorID = 19387 THEN
			stDriveInfo.DeviceType := E_DeviceType.DEVICETYPE_UNKNOWN;
			nSeq := 20;
		ELSIF fbReadDriveType.Error THEN
			nSeq := nSeq + 1000;
		ELSIF NOT fbReadDriveType.Busy THEN
			stDriveInfo := fbReadDriveType.DriveInfo;
			nSeq := 20;
		END_IF
		
	20: //Delete current NC2 Offset	
		fbSetPosNC.Options.ClearPositionOffset 	:= TRUE;
		fbSetPosNC.Execute 						:= TRUE; 
		nSeq := 21;

	21: //Delete current NC2 Offset	
		IF fbSetPosNC.Error THEN
			nSeq := nSeq + 1000;
		ELSIF NOT fbSetPosNC.Busy THEN
			fbSetPosNC.Execute								:= FALSE; 
			fbSetPosNC.Options.ClearPositionOffset 	:= FALSE;
			nSeq := 30;
		END_IF	
		
	30: //Execute CoE/SoE read to get selectet store mode (Drive, Encoder)
		CASE stDriveInfo.DeviceType OF
			//ELM
			DEVICETYPE_ELM72xx_OCT, DEVICETYPE_ELM72xx_OCT_SAFETY:
				fbCoERead.Execute				:= TRUE; 
				IF stDriveInfo.Channel = 0 THEN
					fbCoERead.Index				:= 16#8000;
					fbCoERead.SubIndex			:= 16#0D; 
				ELSIF stDriveInfo.Channel = 1 THEN
					fbCoERead.Index				:= 16#8100;
					fbCoERead.SubIndex			:= 16#0D; 
				END_IF


			//AX80xx
			DEVICETYPE_AX8000:                    	
				fbCoERead.Execute				:= TRUE; 
				IF stDriveInfo.Channel = 0 THEN
					fbCoERead.Index				:= 16#3007;
					fbCoERead.SubIndex			:= 16#02;  
				ELSIF stDriveInfo.Channel = 1 THEN
					fbCoERead.Index				:= 16#3407;
					fbCoERead.SubIndex			:= 16#02; 
				END_IF
				
				
			//EL72xx 
			DEVICETYPE_EL72x1, DEVICETYPE_EL72x1_OCT, DEVICETYPE_EL72x1_OCT_SAFETY:
				;//EL72xx does not support save in encoder memory
	
				
			//AX50xx	
			DEVICETYPE_SOE_DEFAULT: 
				fbSoERead.Execute			:= TRUE;        	
				fbSoERead.Idn				:= (P_0_IDNs + 275);
				fbSoeRead.Element 			:= 16#40;//the value of the parameter
				
			//Unknown or virtual	
     		ELSE
				;
		END_CASE
		nSeq := 40;
		
		
	40: //Write E_PositionOffsetMemory 
		CASE stDriveInfo.DeviceType OF
			//ELM
			DEVICETYPE_ELM72xx_OCT, DEVICETYPE_ELM72xx_OCT_SAFETY:
				IF fbCoERead.Error THEN
					nSeq := nSeq + 1000;
				ELSIF NOT fbCoERead.Busy THEN
					(*	Enum Value	Description
						2 (0x02)	drive_memory
						1 (0x01)	encoder_memory
						0 (0x00)	offset_disabled	*)
					bSetOffsetInNC := (eReadFromCoe = 0);
					fbSetPositionOffset.Memory  := UINT_TO_BYTE(eReadFromCoe - 1);	
					nSeq := 50;
				END_IF

				
			//AX80xx
			DEVICETYPE_AX8000:                    	
				IF fbCoERead.Error THEN
					nSeq := nSeq + 1000;
				ELSIF NOT fbCoERead.Busy THEN
					(*	CH1:3007:04 CH2:3407:04 Offset additional position actual value source 
					https://infosys.beckhoff.com/content/1033/ax8xxx_object/8598064523.html 
						Enum Value	Description
						2 (0x02)	drive_memory
						1 (0x01)	encoder_memory
						0 (0x00)	offset_disabled	 *)
					bSetOffsetInNC := (eReadFromCoe = 0);
					fbSetPositionOffset.Memory  := UINT_TO_BYTE(eReadFromCoe - 1);
					nSeq := 50;
				END_IF
				
				
			//EL72xx 
			DEVICETYPE_EL72x1, DEVICETYPE_EL72x1_OCT, DEVICETYPE_EL72x1_OCT_SAFETY:
				//EL72xx does not support save in encoder memory
				fbSetPositionOffset.Memory := E_PositionOffsetMemory.ePositionOffsetMemory_Drive;
				nSeq := 50;
				
			//AX50xx	
			DEVICETYPE_SOE_DEFAULT: 
				IF fbSoERead.Error THEN
					nSeq := nSeq + 1000;
				ELSIF NOT fbCoERead.Busy THEN
					(*	P-0-0275-Position offset control / Feedback 1
					https://infosys.beckhoff.com/content/1033/ax5000_idn_description/1365901707.html
						Enum Value	Description
						2 (0x02)	drive_memory
						1 (0x01)	encoder_memory
						0 (0x00)	offset_disabled		*)
					bSetOffsetInNC := (eReadFromSoE = 0);
					fbSetPositionOffset.Memory := UINT_TO_BYTE(eReadFromSoE - 1);
					nSeq := 50;
				END_IF
				
			//Unknown or virtual	
     		ELSE
				bSetOffsetInNC := TRUE;
				nSeq := 50;
		END_CASE
			
		
	50:	//Decide whether Nc should be stored 
		//temporarily in the NC or permanently in the drive/encoder
		IF bSetOffsetInNC THEN
			THIS^.bStoredInNc := TRUE;
			nSeq := 100;
		ELSE
			THIS^.bStoredInDrive := fbSetPositionOffset.Memory = E_PositionOffsetMemory.ePositionOffsetMemory_Drive;
			THIS^.bStoredInEncoder := fbSetPositionOffset.Memory = E_PositionOffsetMemory.ePositionOffsetMemory_Encoder;
			nSeq := 200;
		END_IF

	
	100://Set offset in NC	
		fbSetPosNC.Execute	:= TRUE; 
		fbSetPosNC.Position	:= THIS^.fPosition; 
		fbSetPosNC.Mode		:= THIS^.bMode; (* RELATIVE=True, ABSOLUTE=False*)	
		nSeq := 101;
		
	101: // DONE
		THIS^.Done			:= fbSetPosNC.Done;
		THIS^.Busy			:= fbSetPosNC.Busy;
		THIS^.Error			:= fbSetPosNC.Error;
		THIS^.ErrorID 		:= fbSetPosNC.ErrorID;	

	200://Delete current offset in NC	
		fbDeletePositionOffset.Execute	:= TRUE; 
		fbDeletePositionOffset.Feedback	:= E_PositionOffsetFeedback.ePositionOffsetFeedback1;
		fbDeletePositionOffset.Memory	:= fbSetPositionOffset.Memory;
		nSeq := 201;		
		
	201://Delete current offset in NC
		IF fbDeletePositionOffset.Error THEN
			nSeq := nSeq + 1000;
		ELSIF NOT fbDeletePositionOffset.Busy THEN
			nSeq := 202;
		END_IF	
		
	202://Set offset in Drive/Encoder	
		fbSetPositionOffset.Execute		:= TRUE; 
		fbSetPositionOffset.Position	:= THIS^.fPosition; 
		fbSetPositionOffset.Relative	:= THIS^.bMode; (* RELATIVE=True, ABSOLUTE=False*)	
		fbSetPositionOffset.Feedback	:= E_PositionOffsetFeedback.ePositionOffsetFeedback1;
		fbSetPositionOffset.Memory		:= fbSetPositionOffset.Memory;
		nSeq := 203;
		
	203: // DONE
		THIS^.Done			:= (NOT fbSetPositionOffset.Busy) AND (NOT fbSetPositionOffset.Error) ;
		THIS^.Busy			:= fbSetPositionOffset.Busy;
		THIS^.Error			:= fbSetPositionOffset.Error;
		THIS^.ErrorID 		:= fbSetPositionOffset.ErrorID;	
		
	1000..1999: //Error
		THIS^.Done			:= FALSE;
		THIS^.Busy			:= FALSE;
		THIS^.Error			:= TRUE;
		THIS^.ErrorID 		:= nSeq;
		
END_CASE	

//Cyclic update
fbCoERead(Axis:= THIS^.Axis, pDstBuf := ADR(eReadFromCoe), BufLen := SIZEOF(eReadFromCoe));
fbSoERead(Axis:= THIS^.Axis, pDstBuf := ADR(eReadFromSoE), BufLen := SIZEOF(eReadFromSoE));
fbReadDriveType(Axis := Axis);
fbSetPositionOffset(Axis := Axis);
fbSetPosNC(Axis := Axis);

END_FUNCTION_BLOCK

// COMPONENTs/Optional/Adapter HMI/FB_NcAxis_Hmi
FUNCTION_BLOCK FB_NcAxis_Hmi
VAR
    {attribute 'hide'}
    ipAxis : I_NcAxis_HMI;
    {attribute 'hide'}	
	bValidInterface : BOOL;

    fPosition     	: LREAL;
    fVelocity     	: LREAL;
    fAcceleration 	: LREAL;
	bMoving		  	: BOOL;
    bCoupled      	: BOOL;
	bError      	: BOOL;
	bBusy      		: BOOL;
	bDone      		: BOOL;
	sLUID			: STRING;		//Locally unique identifier
	sNcAxisName		: STRING(31);
	sState       	: STRING(20);
END_VAR

VAR CONSTANT
	{attribute 'hide'}
	//List of string of axis states
	AXIS_STATES: ARRAY[0..8] OF STRING(20) := [	'UNDEFINED',
												'DISABLED',
												'STANDSTILL',
												'ERRORSTOP',
												'STOPPING',
												'HOMING',
												'DISCRETEMOTION',
												'CONTINOUSMOTION',
												'SYNCHRONIZEDMOTION'];
END_VAR

METHOD FB_init : BOOL
VAR_INPUT
	bInitRetains : BOOL; // if TRUE, the retain variables are initialized (warm start / cold start)
	bInCopyCode : BOOL;  // if TRUE, the instance afterwards gets moved into the copy code (online change)
	
	ipAxis : I_NcAxis_HMI;
END_VAR
VAR_INST
	{attribute 'hide'}
	bFBInitCalledOnce : BOOL; //Do the following code once during start up and not during onlinechange
END_VAR
//Do the following code once during start up and not during onlinechange
IF NOT bFBInitCalledOnce THEN 
	THIS^.ipAxis := ipAxis;
	THIS^.bValidInterface := THIS^.ipAxis <> 0;
END_IF

bFBInitCalledOnce := TRUE;
END_METHOD

METHOD Update : HRESULT
VAR_INPUT
END_VAR
IF NOT THIS^.bValidInterface THEN
	//Error, no valide interface
	Update := E_FAIL;
	RETURN;
END_IF


//Convert data from interface to local variables
fPosition     	:=THIS^.ipAxis.SetPosition;
fVelocity     	:=THIS^.ipAxis.SetVelocity;
fAcceleration 	:=THIS^.ipAxis.SetAcceleration;
bCoupled      	:=THIS^.ipAxis.Coupled;
bMoving     	:=THIS^.ipAxis.Moving;
bError      	:=THIS^.ipAxis.Feedback.Error;
bBusy      		:=THIS^.ipAxis.Feedback.Busy;
bDone      		:=THIS^.ipAxis.Feedback.Done;
sLUID			:=THIS^.ipAxis.LUID;
sNcAxisName		:=THIS^.ipAxis.NcAxisName;
sState			:=THIS^.AXIS_STATES[THIS^.ipAxis.MotionState];
END_METHOD

END_FUNCTION_BLOCK

// COMPONENTs/Optional/Casting/ToNcAxisHMI
FUNCTION ToNcAxisHMI : BOOL
VAR_INPUT
	ipChObject : I_CH_OBJECT;
	ipNcAxisHMI : REFERENCE TO I_NcAxis_HMI;
END_VAR

VAR
	ipTmp : I_NcAxis_HMI;
END_VAR

(* 
   1. Test if the interface exists
   2. Test if the object implements a "Object" interface 
   3. Write reference to interface in parameter
   4. Returne TRUE if succesfull
*)
IF ipChObject <> 0 AND_THEN __QUERYINTERFACE(ipChObject,ipTmp) THEN
	ipNcAxisHMI := ipTmp;
	ToNcAxisHMI := TRUE;
END_IF

END_FUNCTION

// COMPONENTs/Optional/Casting/ToNcAxisPLC
FUNCTION ToNcAxisPLC : BOOL
VAR_INPUT
	ipChObject : I_CH_OBJECT;
	ipNcAxisPLC : REFERENCE TO I_NcAxis_PLC;
END_VAR

VAR
	ipTmp : I_NcAxis_PLC;
END_VAR

(* 
   1. Test if the interface exists
   2. Test if the object implements a "Object" interface 
   3. Write reference to interface in parameter
   4. Returne TRUE if succesfull
*)
IF ipChObject <> 0 AND_THEN __QUERYINTERFACE(ipChObject,ipTmp) THEN
	ipNcAxisPLC := ipTmp;
	ToNcAxisPLC := TRUE;
END_IF

END_FUNCTION

// COMPONENTs/Optional/SetActPosition/old/FB_SetPosition_NC_Sercos_CANopen
{attribute 'hide_all_locals'}
FUNCTION_BLOCK FB_SetPosition_NC_Sercos_CANopen
VAR_INPUT
    Execute  : BOOL;
    Position : LREAL; 
    Mode     : BOOL; // RELATIVE=True, ABSOLUTE=False (Default)
    //Options  : ST_SetPositionOptions; // only Feedback1 is supportet
END_VAR

VAR_OUTPUT
    Done    : BOOL;
    Busy    : BOOL;
    Error   : BOOL;
    ErrorID : UDINT;
END_VAR

VAR_IN_OUT
    Axis 	: AXIS_REF;
END_VAR

VAR 
	fPosition 			: LREAL;
	bMode     			: BOOL; // RELATIVE=True, ABSOLUTE=False (Default)
	nSeq 				: UDINT :=0;
	nSeqCoE 			: UDINT :=0;
	nSeqSoE				: UDINT :=0;
	nSeqNC 				: UDINT :=0;
	
	fbTriggerExecute	: R_TRIG;
	
	fbReadDriveAddress 	: MC_ReadDriveAddress;
	fbSetPosNC 			: MC_SetPosition;
	fbSetPosAX5xxx		: FB_SoEAX5000SetPositionOffset;
	fbSetPosAX8xxx		: FB_CoEAX8000SetPositionOffset;
	fbSetPosEL72xxx		: FB_CoEEL72xxSetPositionOffset;
	fbCoERead 			: FB_CoERead;
	fbSoERead 			: FB_SoERead;
	fbAdsWrite			: ADSWRITE;
	strDeviceName		: STRING;
	
	
	eReadPositionOffsetMemory    : E_PositionOffsetMemory;
	eReadFromCoe :UINT := 99;
	eReadFromSoe :UINT := 99;
END_VAR

fbTriggerExecute(CLK:= THIS^.Execute);
//Reset on positive execution edge
IF fbTriggerExecute.Q THEN
	THIS^.Done	:= FALSE;
	THIS^.Busy	:= TRUE;
	THIS^.Error	:= FALSE;
	nSeqCoE		:= 0;
	nSeqSoE		:= 0;
	nSeqNC		:= 0;
	bMode 		:= Mode;
	fPosition 	:= Position;
END_IF

IF NOT (THIS^.Busy OR THIS^.Execute) THEN
	THIS^.Done			:=FALSE;
	THIS^.Busy			:=FALSE;
	THIS^.Error			:=FALSE;
	THIS^.ErrorID 		:= 0;
	nSeqCoE				:= 0;
	nSeqSoE				:= 0;
	nSeqNC				:= 0;
	fbReadDriveAddress.Execute := FALSE;
END_IF

	
//call update methode during execution
IF THIS^.Busy THEN
	CASE THIS^.Axis.DriveAddress.NcDriveType OF 
		//Sercos
		Tc2_MC2.E_NcDriveType.NcDriveType_Sercos:
			SetPosSoE();
			
		//MDP742 (Ax8000, EL72xx,...)
		Tc2_MC2.E_NcDriveType.NcDriveType_CANopen_DS402_MDP742:
			SetPosCoE();	
		
		//Undefined. Do an MC_ReadDriveAddress first.
		Tc2_MC2.E_NcDriveType.NcDriveType_undefined:	
			fbReadDriveAddress.Execute := TRUE;
			IF fbReadDriveAddress.Done THEN
				Axis.DriveAddress := fbReadDriveAddress.DriveAddress;
			END_IF

		//Simulation or not supported axis	
		ELSE
			SetPosNC();				
	END_CASE
END_IF

		

fbReadDriveAddress(Axis := Axis);

METHOD PRIVATE SetPosCoE : HRESULT
VAR_INPUT
END_VAR
// The warning " Access to VAR_IN_OUT..." can be disabled here. This Methode is private and so only called if the FB IN_OUT_VAR is valid
{warning disable C0371}

CASE nSeqCoE OF
	0:	// **********************  Init *****************************************
		fbSetPosAX8xxx.Execute		:= FALSE;
		fbSetPosEL72xxx.Execute		:= FALSE;
		fbCoERead.Execute			:= FALSE; 
		fbAdsWrite.WRITE			:= FALSE;
		nSeqCoE := 10;
	
	10: // ********************** SetPosition is only posible if axis is disabled **********************
		IF NOT THIS^.Axis.Status.StandStill THEN
			nSeqCoE := nSeqCoE + 1000;
		ELSE
			nSeqCoE := 50;	
		END_IF
		
	50: // ********************** Re-initialization of the actual NC-encoder position **********************
		// IF in the Nc is an Offset active (SetPos or MC_Home) then the calculated offset for the Encoder oder Drive is wrong.
		fbAdsWrite.WRITE			:= TRUE;
		fbAdsWrite.PORT				:= 501; //NC-Port
		fbAdsWrite.IDXGRP			:= (16#5200 + THIS^.Axis.NcToPlc.AxisId);//"Index offset" specification for encoder functions (Index group 0x5200 + ID)
		fbAdsWrite.IDXOFFS			:= 16#1B; //https://infosys.beckhoff.com/content/1033/tc3_ads_intro/713106315.html 
		fbAdsWrite.LEN				:= 0; //VOID
		fbAdsWrite.SRCADDR			:= 0; //VOID
		nSeqCoE := 60;

	60: // ********************** wait for Re-initialization of the actual NC-encoder position **********************
		IF fbAdsWrite.ERR THEN
			nSeqCoE := nSeqCoE + 1000;
		ELSIF NOT fbAdsWrite.Busy THEN
			fbAdsWrite.WRITE := FALSE;
			nSeqCoE := 110;				
		END_IF
	

			
	110:// **********************  Coe Read Device Name to decide *****************************************	
		fbCoERead.Execute			:= TRUE; 
		fbCoERead.Index				:= 16#1008;
		fbCoERead.SubIndex			:= 0; 
		fbCoERead.pDstBuf			:= ADR(strDeviceName);
		fbCoERead.BufLen			:= SIZEOF(strDeviceName);
		nSeqCoE := 120;
 		
